// TIA Portal project "SortingStantion" (V16)
// Станция сортировки и отбраковки

(* hardware
DEVICE "S7-1200 station_1"  S7-1200 Station
   slot 0: "Rack_0"  S7-1200 Rack  Rack  V1.0
   slot 1: "6ES7 214-1AG40-0XB0"  CPU 1214C DC/DC/DC  6ES7 214-1AG40-0XB0  V4.4
*)

// ===== PLC "6ES7 214-1AG40-0XB0"  CPU 1214C DC/DC/DC =====

VAR_GLOBAL   // PLC tag table "Default tag table"
   "sensorFS1" AT %I200.0 : Bool;   // Фотодатчик 1
   "Tag_4" AT %IW0 : Word;
   "FS1" AT %I0.0 : Bool;   // Фотодатчик 1 (перед сканером)
   "GOOD_READ_SIGNAL" AT %I0.4 : Bool;   // Сигнал goodread
   "NO_READ_SIGNAL" AT %I0.3 : Bool;   // Сигнал NO_READ
   "FS2" AT %I0.1 : Bool;   // Фотодатчик перед отбраковщиком
   "FS3" AT %I0.2 : Bool;   // Фотодатчик на выходе отбраковщика
   "UPS_OK" AT %I0.5 : Bool;   // Статус ИБП - ОК
   "Conveyor_ON_impulse" AT %Q0.6 : Bool;
   "SCANER_PHASE_ON" AT %Q0.0 : Bool;   // Сингал для начала фазы сканирования
   "GreenLamp" AT %Q0.3 : Bool;
   "RedLamp" AT %Q0.4 : Bool;
   "PUSHER_OUT" AT %Q0.2 : Bool;
   "Buzzer" AT %Q0.5 : Bool;
   "Tag_6" AT %QW0 : Word;
   "SCANER_PHASE_OFF" AT %Q0.1 : Bool;   // Сигнал для окончания фазы сканирования
   "Conveyor_OFF_impulse" AT %Q0.7 : Bool;
   "Conveyor_ON_duplicate" AT %Q1.1 : Bool;
   "Tag_1" AT %M10.0 : Bool;
   "photoSensor0" AT %M0.0 : Bool;
   "sensorFS2" AT %M0.1 : Bool;
   "sensorFS3" AT %M0.2 : Bool;
   "System_Byte" AT %MB10 : Byte;
   "DiagStatusUpdate" AT %M10.1 : Bool;
   "AlwaysTRUE" AT %M10.2 : Bool;
   "AlwaysFALSE" AT %M10.3 : Bool;
   "Tag_2" AT %M2.0 : Bool;
   "Tag_3" AT %MD100 : DWord;
   "Tag_5" AT %MW0 : Word;
   "GoodRead" AT %M0.3 : Bool;
   "NoRead" AT %M0.4 : Bool;
   "Tag_7" AT %M1.3 : Bool;
   "Tag_8" AT %M1.4 : Bool;
   "FP_NEW_TASK" AT %M1.0 : Bool;
   "System" AT %M8.0 : Bool;
   "FN_MAIN_INTLK" AT %M8.1 : Bool;
   "FP_PHASE_ON" AT %M8.2 : Bool;
   "GoodReadTSignal" AT %M3.0 : Bool;
   "NoReadTSignal" AT %M3.1 : Bool;
   "wBuffer" AT %MW4 : Word;
   "HiChar" AT %MB4 : Byte;
   "loChar" AT %MB5 : Byte;
   "MEMMORYCELL_PRODUCT_DEFFECT_SETPOINT" AT %MD0 : DWord;
   "Tag_9" AT %M5.0 : Bool;
   "StrobeMerker" AT %M8.3 : Bool;
   "Control_begin" AT %M200.1 : Bool;   // Флаг запуска процесса контроля отбраковки
   "Tag_12" AT %M200.0 : Bool;
   "Tag_10" AT %MD170 : DInt;
   "TestMode" AT %M13.0 : Bool;
   "Clock_Byte" AT %MB65 : Byte;
   "Clock_10Hz" AT %M65.0 : Bool;
   "Clock_5Hz" AT %M65.1 : Bool;
   "Clock_2.5Hz" AT %M65.2 : Bool;
   "Clock_2Hz" AT %M65.3 : Bool;
   "Clock_1.25Hz" AT %M65.4 : Bool;
   "Clock_1Hz" AT %M65.5 : Bool;
   "Clock_0.625Hz" AT %M65.6 : Bool;
   "Clock_0.5Hz" AT %M65.7 : Bool;
   "Tag_14" AT %M13.1 : Bool;
   "Tag_15" AT %M13.2 : Bool;
   "Tag_16" AT %M13.3 : Bool;
   "Tag_17" AT %M13.4 : Bool;
   "Tag_19" AT %M64.0 : Bool;
   "Tag_20" AT %M13.5 : Bool;
   "Tag_21" AT %MB14 : Byte;
   "Tag_22" AT %MD14 : DWord;
   "Tag_23" AT %MD22 : DWord;
   "Tag_24" AT %M13.7 : Bool;
   "Tag_25" AT %MB11 : Byte;
   "Tag_26" AT %M13.6 : Bool;
   "Tag_27" AT %M198.6 : Bool;
   "Tag_11" AT %M8.4 : Bool;
   "FP_ERR_TRANSMITION" AT %M8.5 : Bool;
   "Tag_13" AT %M25.0 : Bool;
   "Tag_28" AT %M25.1 : Bool;
   "Флаг начала работы толкателя" AT %M25.2 : Bool;
   "Conveyor_ON" AT %Q1.0 : Bool;
END_VAR

TYPE "PRODUCT"
VERSION : 0.1
   STRUCT
      IS_ACTUAL : Bool := false;   // Флаг, указывающий на актуальность данных
      IS_GOOD : Bool;   // Флаг, указывающий то, что отбраковка не нужна
      ID : UDInt;   // Позиция в очереди
      BARCODE : String[100];   // Штрихкод из сканера в виде массива байт
      "TIME" : DTL;   // Метка времени
   END_STRUCT;
END_TYPE

DATA_BLOCK "GlobalData"   // DB1
{ S7_Optimized_Access := 'FALSE' }
VERSION : 0.1
   VAR
      INTERLOCK : Struct
         RESET_COUNTER_DISCONNECT : Bool;   // Команда для сброса счетчика, определяющего потерб связи с ПК
         MAIN_INTERLOCK : Bool;   // Главная деблокировка
         ACTIVE_ALARMS : Bool;   // Флаг, указывающий на наличае хотя бы одной ошибки
         DISCONNECT_COUNTER : UInt;   // Счетчик, по которому определяется потеря связи с ПК
         SPARE : Array[0..10] of Byte;
      END_STRUCT;
      AUX : Struct
         COUNTERS : Struct   // Счетчики заготовок
            QUANTITY_PRODUCTS : UDInt;   // Общее количество изделий, пройденых по конвейеру
            QUANTITY_BOXS : UDInt;   // Счетчик коробов
            QUANTITY_PRODUCTS_AUTO_REJECTED : UDInt;   // Количество изделий, отбракованых отбраковщиком автоматически
            QUANTITY_PRODUCTS_MANUAL_REJECTED : UDInt;   // Количество изделий, отбракованых вручную
            DEFECT_COUNTER : UDInt;   // Счетчик дефектного продукта
            REPEAT_COUNTER : UDInt;   // Счетчик повторов кодов
            SPARE : Array[0..22] of Word;
         END_STRUCT;
         BUZZER_ACTIVATE : Bool;   // Флаг активации звукового извещателя
         CONVEYOR_IS_STOPPED : Bool;   // Флаг, указывающий, что конвейер остановлен
         SPARE : Array[0..9] of Byte;
      END_STRUCT;
      FROM_HMI : Struct
         CTW : Struct   // Слово управления
            AUX_RUN_CMD : Bool;   // Команда для работы из PC
            RESET_ALARMS_CMD : Bool;   // Команда для сброса ошибок
            CLER_COLLECTION_CMD : Bool;   // Команда для очистки очереди изделий между отбраковщиком и сканером
            SIM_MODE_ACTIVE : Bool;   // Команда для активации режима симуляции
            CONVEYOR_FORCE_RUN : Bool;   // Команда для принудительного запуска конвейера
            HMI_IS_RUN : Bool;
            RUN_CMD_FROM_HMI : Bool;
            SPARE : Byte;
         END_STRUCT;
         SETTINGS : Struct   // Настройки панели
            IGNORE_REPEAT_PRODUCT_CODE_1 : Bool;   // Команда для игнорирования повтора кода продукта
            TIME_A : Time := T#5s;   // Задержка включения сканера, ms
            TIME_B : Time := T#5s;   // Длительность фазы чтения штрихкода, ms
            TIME_C : Time := T#5s;   // Время ожидания результа от сканера
            TIME_D : Time := T#4s;   // Длительность фазы чтения штрихкода, ms
            TIME_PUSHER_ACTIVE : Time := T#5s;   // Длительность импульса толкателя
            TIME_E : Time := T#5s;   // Время контроля отбраковки
            STOP_DELAY : Time := T#5s;   // Задержка остановки
            PRODUCT_DEFFECT_SETPOINT : UDInt := 5;   // Массовый брак (уставка)
            IGNORE_REPEAT_PRODUCT_CODE : Bool;   // Команда для игнорирования повтора кода продукта
            DEAD_TIME : Time := T#0ms;
            SPARE : Array[0..6] of Byte;
         END_STRUCT;
         CURRENT_TASK : Struct   // Текущее задание
            IN_WORK : Bool;   // Флаг, указывающий, что задание нахожится в работе
            ID : String[40];   // Уникальный идентификатор задания
            GTIN : String[40];   // Номер GTIN. (14 символов)
            PRODUCT_NAME : String[82];   // Наименование продукта
            LOT_NO : String[40];   // Номер производственной серии (до 20 символов)
            LINE_NUM : UInt := 0;   // Номер линии для, которой сформировано это задание.
            NUM_PACKS_IN_BOX : UDInt := 0;   // Кол-во продуктов в коробе.
            NUM_PACKS_IN_SERIES : UDInt := 0;   // Ожидаемое количество продуктов в серии (определяется по заданию на производство серии)
         END_STRUCT;
         SPARE : Array[0..6] of Byte;
      END_STRUCT;
      TO_HMI : Struct
         READ_PRODUCT_CMD : Bool;   // Команда для считывания данных продукта
      END_STRUCT;
      PRODUCT_IS_SCANING_AREA : "PRODUCT";   // Продукт в зоне сканирования
      PRODUCT_IS_PUSHER_AREA : "PRODUCT";   // Продукт в зоне отбраковки
      RESULT_STR : String;
      RCV_PRODUCT_ID : UDInt;   // ID продукта, полученного из L2 rкак подтверждение получения
   END_VAR
BEGIN
END_DATA_BLOCK

// folder: 10_ForTest

DATA_BLOCK "TestCodesGenerate_DB"   // DB25
{ S7_Optimized_Access := 'TRUE' }
VERSION : 0.1
// stored: InstanceOfName TestCodesGenerate
"TestCodesGenerate"
BEGIN
END_DATA_BLOCK

DATA_BLOCK "TestDB"   // DB26
{ S7_Optimized_Access := 'TRUE' }
VERSION : 0.1
   VAR
      Test_products : Array[0..1] of String[10];
      Test_disable_flag : Bool;
      Index_for_testproduct : UDInt;
      Actual_testproduct : String[50];
      counter_transfer_products : UDInt;
   END_VAR
BEGIN
   // Test_products[0] : Test_products
END_DATA_BLOCK

// folder: 2_КОНВЕЙЕР

DATA_BLOCK "CONVEYOR_DB"   // DB3
{ S7_Optimized_Access := 'TRUE' }
VERSION : 0.1
// stored: InstanceOfName CONVEYOR
"CONVEYOR"
BEGIN
END_DATA_BLOCK

// folder: 4_СКАНЕР MATRIX

DATA_BLOCK "SCANER_DB"   // DB2
{ S7_Optimized_Access := 'FALSE' }
VERSION : 0.1
// stored: InstanceOfName mSCANER
"mSCANER"
BEGIN
END_DATA_BLOCK

DATA_BLOCK "MODBUS_DATA"   // DB9
{ S7_Optimized_Access := 'FALSE' }
VERSION : 0.1
   VAR
      TCP_CONNECTION : TCON_IP_v4;
      MODBUS_DATA : Array[0..100] of Word;
      BYTES_ARRAY : Array[0..200] of Byte;
      Scaner_not_connected : Bool;
   END_VAR
BEGIN
   TCP_CONNECTION.ConnectionType := 11;
   TCP_CONNECTION.ID := 3;
   TCP_CONNECTION.InterfaceId := 64;
   TCP_CONNECTION.LocalPort := 502;
   TCP_CONNECTION.RemoteAddress.ADDR[1] := 0;
   TCP_CONNECTION.RemoteAddress.ADDR[2] := 0;
   TCP_CONNECTION.RemoteAddress.ADDR[3] := 0;
   TCP_CONNECTION.RemoteAddress.ADDR[4] := 0;
END_DATA_BLOCK

// folder: 5_ОТБРАКОВЩИК

DATA_BLOCK "PUSHER_CONTROL_DB"   // DB4
{ S7_Optimized_Access := 'TRUE' }
VERSION : 0.1
// stored: InstanceOfName PUSHER_CONTROL
"PUSHER_CONTROL"
BEGIN
END_DATA_BLOCK

DATA_BLOCK "PUSHER_DB_1"   // DB22
{ S7_Optimized_Access := 'TRUE' }
VERSION : 0.1
// stored: InstanceOfName PUSHER
"PUSHER"
BEGIN
END_DATA_BLOCK

// folder: 6_КОЛЛЕКЦИЯ ИЗДЕЛИЙ

DATA_BLOCK "ITEMS_COLLECTION"   // DB5
{ S7_Optimized_Access := 'FALSE' }
VERSION : 0.1
   VAR
      PRODUCTS_BEFOR_PUSHER : Struct
         LENGHT : UDInt;   // Количество изделий в коллекции
         INDEX : UDInt;   // Индекс для определения ID
         PRODUCTS : Array[0..20] of "PRODUCT";   // Коллекция невыпущенных продуктов
      END_STRUCT;
      PRODUCTS_IN_SEND_TO_PC : Struct
         LENGHT : UDInt;   // Количество изделий в коллекции
         INDEX : UDInt;   // Индекс для определения ID
         PRODUCTS : Array[0..3] of "PRODUCT";   // Коллекция продуктов в зоне отбраковщика
      END_STRUCT;
   END_VAR
BEGIN
END_DATA_BLOCK

// folder: 7_СООБЩЕНИЯ

DATA_BLOCK "ALARMS"   // DB6
{ S7_Optimized_Access := 'FALSE' }
VERSION : 0.1
   VAR
      WARNINGS : Struct
         WARNINGS_W0 : Word;   // Тэг для HMI
         WARNINGS_W1 : Word;   // Тэг для HMI
         WARNING_0_TASK_NOT_ACCEPTED : Bool;   // Сообщение - Задача не принята
         spare_1 : Bool;
         spare_2 : Bool;
         spare_3 : Bool;
         spare_4 : Bool;
         spare_5 : Bool;
         spare_6 : Bool;
         spare_7 : Bool;
         spare_8 : Bool;
         spare_9 : Bool;
         spare_10 : Bool;
         spare_11 : Bool;
         spare_12 : Bool;
         spare_13 : Bool;
         spare_14 : Bool;
         spare_15 : Bool;
         spare_16 : Bool;
         spare_17 : Bool;
         spare_18 : Bool;
         spare_19 : Bool;
         spare_20 : Bool;
         spare_21 : Bool;
         spare_22 : Bool;
         spare_23 : Bool;
         spare_24 : Bool;
         spare_25 : Bool;
         spare_26 : Bool;
         spare_27 : Bool;
         spare_28 : Bool;
         spare_29 : Bool;
         spare_30 : Bool;
         spare_31 : Bool;
      END_STRUCT;
      ALARMS : Struct
         ALARMS_W0 : Word;   // Тэг для HMI
         ALARMS_W1 : Word;   // Тэг для HMI
         ERROR_1_FS1_FAULT : Bool;   // Неисправность фотодатчика 1
         ERROR_2_FS2_FAULT : Bool;   // Неисправность фотодатчика 2
         ERROR_3_FS3_FAULT : Bool;   // Неисправность фотодатчика 3
         ERROR_4_REPEAT_PRODUCT_CODE : Bool;   // Повтор кода продукта
         ERROR_5_RECEIVING_CODE_WHEN_LINE_STOPS : Bool;   // Получение кода от сканера при остановке конвейера
         ERROR_6_ERROR_PUSHER : Bool;   // Ошибка отбраковщика (продукт не отбраковался)
         ERROR_7_OVER_DEFECT_COUNTER : Bool;   // Массовый брак
         ERROR_8_ERROR_TRANSMITIOM_BARCODE : Bool;   // Ошибка отбраковщика
         ERROR_9_ProductsAreTooCloseToEachOtherRangeScaner : Bool;   // Продукт слишком близко друг к другу
         ERROR_9_ProductsAreTooCloseToEachOtherRangePusher : Bool;
         ERROR_11_SPARE : Bool;
         ERROR_NO_TASK : Bool;   // Ошибка - нет принятой задачи
         ERROR_POWER_SYPLE : Bool;   // Ошибка питания (по сигналу от ИБП)
         ERROR_12_AutoScaner_NotConnected : Bool;
         spare_12 : Bool;
         spare_13 : Bool;
         spare_14 : Bool;
         spare_15 : Bool;
         spare_16 : Bool;
         spare_17 : Bool;
         spare_18 : Bool;
         spare_19 : Bool;
         spare_20 : Bool;
         spare_21 : Bool;
         spare_22 : Bool;
         spare_23 : Bool;
         spare_24 : Bool;
         spare_25 : Bool;
         spare_26 : Bool;
         spare_27 : Bool;
         spare_28 : Bool;
         spare_29 : Bool;
      END_STRUCT;
   END_VAR
BEGIN
END_DATA_BLOCK

// folder: 8_BUZZER

DATA_BLOCK "xBuzzer_DB"   // DB10
{ S7_Optimized_Access := 'TRUE' }
VERSION : 0.1
// stored: InstanceOfName xBuzzer
"xBuzzer"
BEGIN
END_DATA_BLOCK

// folder: 9_PINOUT

DATA_BLOCK "IO"   // DB15
{ S7_Optimized_Access := 'FALSE' }
VERSION : 0.1
   VAR
      INPUTS : Struct
         FS1 : Bool;
         FS2 : Bool;
         FS3 : Bool;
         GoodRead : Bool;
         NoRead : Bool;
         spare : Byte;
      END_STRUCT;
      OUTPUTS : Struct
         mScanerPhaseOn : Bool;
         mScanerPhaseOff : Bool;
         Pusher : Bool;
         GreenLamp : Bool;
         RedLamp : Bool;
         Buzzer : Bool;
         Conveyor : Bool;
         spare : Byte;
      END_STRUCT;
      SIMULATION : Struct
         FS1 : Bool;
         FS2 : Bool;
         FS3 : Bool;
         GoodRead : Bool;
         NoRead : Bool;
         spare : Byte;
      END_STRUCT;
   END_VAR
BEGIN
END_DATA_BLOCK

// folder: System blocks/Program resources

DATA_BLOCK "SDTIMER_ALARM_FS1"   // DB7
{ S7_Optimized_Access := 'TRUE' }
AUTHOR : Simatic
FAMILY : IEC
NAME : IEC_TMR
VERSION : 1.0
// stored: InstanceOfName IEC_TIMER
"IEC_TIMER"
BEGIN
END_DATA_BLOCK

DATA_BLOCK "SDTIMER_ALARM_FS2"   // DB11
{ S7_Optimized_Access := 'TRUE' }
AUTHOR : Simatic
FAMILY : IEC
NAME : IEC_TMR
VERSION : 1.0
// stored: InstanceOfName IEC_TIMER
"IEC_TIMER"
BEGIN
END_DATA_BLOCK

DATA_BLOCK "SDTIMER_ALARM_FS3"   // DB12
{ S7_Optimized_Access := 'TRUE' }
AUTHOR : Simatic
FAMILY : IEC
NAME : IEC_TMR
VERSION : 1.0
// stored: InstanceOfName IEC_TIMER
"IEC_TIMER"
BEGIN
END_DATA_BLOCK

DATA_BLOCK "IEC_Timer_0_DGR"   // DB13
{ S7_Optimized_Access := 'TRUE' }
AUTHOR : Simatic
FAMILY : IEC
NAME : IEC_TMR
VERSION : 1.0
// stored: InstanceOfName IEC_TIMER
"IEC_TIMER"
BEGIN
END_DATA_BLOCK

DATA_BLOCK "IEC_Timer_0_NR"   // DB14
{ S7_Optimized_Access := 'TRUE' }
AUTHOR : Simatic
FAMILY : IEC
NAME : IEC_TMR
VERSION : 1.0
// stored: InstanceOfName IEC_TIMER
"IEC_TIMER"
BEGIN
END_DATA_BLOCK

DATA_BLOCK "IEC_TIM_FS3"   // DB16
{ S7_Optimized_Access := 'TRUE' }
AUTHOR : Simatic
FAMILY : IEC
NAME : IEC_TMR
VERSION : 1.0
// stored: InstanceOfName IEC_TIMER
"IEC_TIMER"
BEGIN
END_DATA_BLOCK

DATA_BLOCK "#IEC_TIM_FS1"   // DB17
{ S7_Optimized_Access := 'TRUE' }
AUTHOR : Simatic
FAMILY : IEC
NAME : IEC_TMR
VERSION : 1.0
// stored: InstanceOfName IEC_TIMER
"IEC_TIMER"
BEGIN
END_DATA_BLOCK

DATA_BLOCK "#IEC_TIM_FS2"   // DB18
{ S7_Optimized_Access := 'TRUE' }
AUTHOR : Simatic
FAMILY : IEC
NAME : IEC_TMR
VERSION : 1.0
// stored: InstanceOfName IEC_TIMER
"IEC_TIMER"
BEGIN
END_DATA_BLOCK

DATA_BLOCK "IEC_TIM_PHASEOFF"   // DB19
{ S7_Optimized_Access := 'TRUE' }
AUTHOR : Simatic
FAMILY : IEC
NAME : IEC_TMR
VERSION : 1.0
// stored: InstanceOfName IEC_TIMER
"IEC_TIMER"
BEGIN
END_DATA_BLOCK

DATA_BLOCK "IEC_Timer_0_DB_1"   // DB20
{ S7_Optimized_Access := 'TRUE' }
AUTHOR : Simatic
FAMILY : IEC
NAME : IEC_TMR
VERSION : 1.0
// stored: InstanceOfName IEC_TIMER
"IEC_TIMER"
BEGIN
END_DATA_BLOCK

DATA_BLOCK "SD_TIMER"   // DB21
{ S7_Optimized_Access := 'TRUE' }
AUTHOR : Simatic
FAMILY : IEC
NAME : IEC_TMR
VERSION : 1.0
// stored: InstanceOfName IEC_TIMER
"IEC_TIMER"
BEGIN
END_DATA_BLOCK

DATA_BLOCK "IEC_Timer_0_DB"   // DB23
{ S7_Optimized_Access := 'TRUE' }
AUTHOR : Simatic
FAMILY : IEC
NAME : IEC_TMR
VERSION : 1.0
// stored: InstanceOfName IEC_TIMER
"IEC_TIMER"
BEGIN
END_DATA_BLOCK

DATA_BLOCK "IEC_Timer_0_DB_2"   // DB24
{ S7_Optimized_Access := 'TRUE' }
AUTHOR : Simatic
FAMILY : IEC
NAME : IEC_TMR
VERSION : 1.0
// stored: InstanceOfName IEC_TIMER
"IEC_TIMER"
BEGIN
END_DATA_BLOCK

DATA_BLOCK "ADDR_SEND_UDP"   // DB29
{ S7_Optimized_Access := 'TRUE' }
   VAR
      ConnectionData : TCON_IP_v4;
      ADDR_Send : TADDR_Param;
   END_VAR
BEGIN
   ConnectionData.ID := 1;
   ConnectionData.ConnectionType := 19;
   ConnectionData.InterfaceId := 64;
   ConnectionData.LocalPort := 2000;
   ConnectionData.RemotePort := 0;
   ConnectionData.ActiveEstablished := false;
   ADDR_Send.REM_PORT_NR := 2000;
   ADDR_Send.REM_IP_ADDR[1] := 192;
   ADDR_Send.REM_IP_ADDR[2] := 168;
   ADDR_Send.REM_IP_ADDR[3] := 3;
   ADDR_Send.REM_IP_ADDR[4] := 97;
END_DATA_BLOCK

DATA_BLOCK "_6ES7 214-1AG40-0XB0_Receive_DB"   // DB30
{ S7_Optimized_Access := 'TRUE' }
   VAR
      ConnectionData : TCON_IP_v4;
      ADDR_Send : TADDR_Param;
   END_VAR
BEGIN
   ConnectionData.ID := 4;
   ConnectionData.ConnectionType := 19;
   ConnectionData.InterfaceId := 64;
   ConnectionData.LocalPort := 2002;
   ConnectionData.RemotePort := 0;
   ConnectionData.ActiveEstablished := false;
   ADDR_Send.REM_PORT_NR := 0;
END_DATA_BLOCK

DATA_BLOCK "ADDR_RCV_UDP"   // DB31
{ S7_Optimized_Access := 'TRUE' }
   VAR
      ConnectionData : TCON_IP_v4;
      ADDR_Send : TADDR_Param;
   END_VAR
BEGIN
   ConnectionData.ID := 2;
   ConnectionData.ConnectionType := 19;
   ConnectionData.InterfaceId := 64;
   ConnectionData.LocalPort := 2001;
   ConnectionData.RemotePort := 0;
   ConnectionData.ActiveEstablished := false;
   ADDR_Send.REM_PORT_NR := 0;
   ADDR_Send.REM_IP_ADDR[1] := 0;
   ADDR_Send.REM_IP_ADDR[2] := 0;
   ADDR_Send.REM_IP_ADDR[3] := 0;
   ADDR_Send.REM_IP_ADDR[4] := 0;
END_DATA_BLOCK

DATA_BLOCK "IEC_Timer_0_DB_3"   // DB32
{ S7_Optimized_Access := 'TRUE' }
AUTHOR : Simatic
FAMILY : IEC
NAME : IEC_TMR
VERSION : 1.0
// stored: InstanceOfName IEC_TIMER
"IEC_TIMER"
BEGIN
END_DATA_BLOCK

// folder: (top level)

ORGANIZATION_BLOCK "Main"   // OB1, LAD, ProgramCycle
TITLE = "Main Program Sweep (Cycle)"
{ S7_Optimized_Access := 'TRUE' }
VERSION : 0.1
   VAR_INPUT
      Initial_Call : Bool;   // Initial call of this OB
      Remanence : Bool;   // =True, if remanent data are available
   END_VAR
   VAR_TEMP
      LineIsRunNormalMode : Bool;   // Флаг, указывающий, что линия запущена в нормальном режиме
      LineRunEnable : Bool;   // Флаг, разрешающий работу линии
      ScanerStage : Word;
      PusherControlStage : Word;
      PusherStage : Word;
   END_VAR
BEGIN

REGION Network 1: Главная деблокировка
   // Проверка разрешения для работы установки
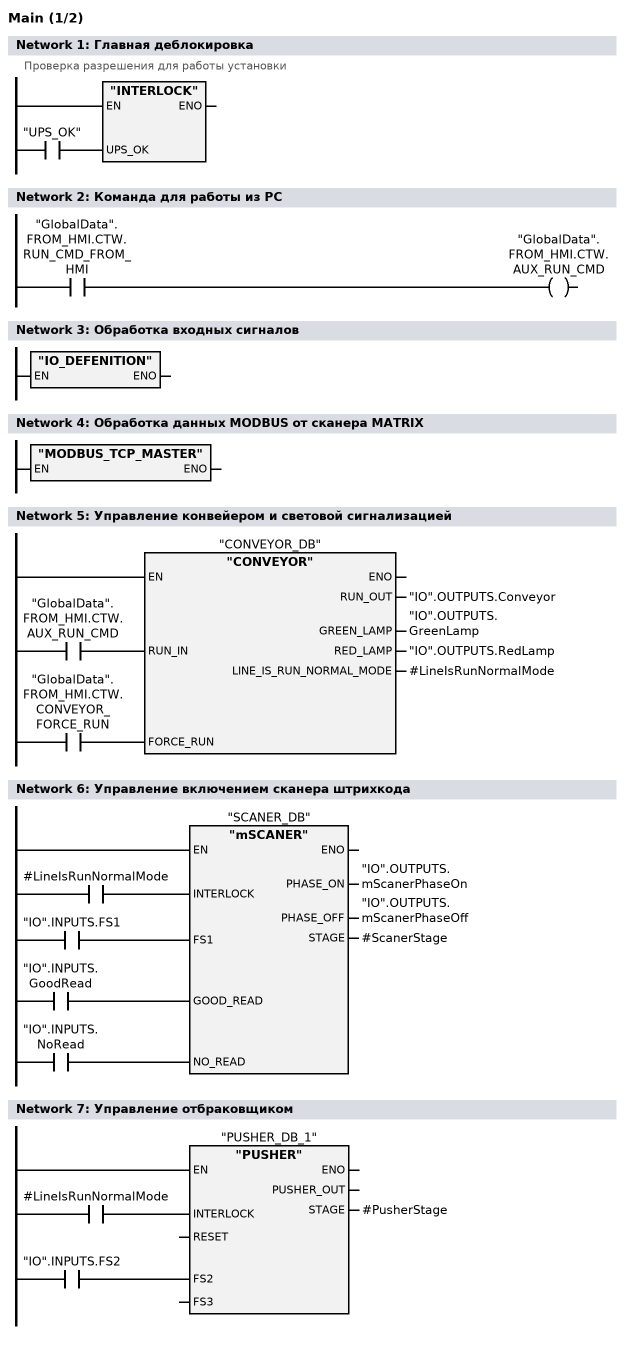
   RUNG wire#powerrail
      "INTERLOCK"(UPS_OK := wire#w1)
   END_RUNG
   RUNG wire#powerrail
      Contact( "UPS_OK" )
   END_RUNG wire#w1
   // the same network as SCL:
   "INTERLOCK"(UPS_OK := "UPS_OK");
END_REGION

REGION Network 2: Команда для работы из PC
   RUNG wire#powerrail
      Contact( "GlobalData".FROM_HMI.CTW.RUN_CMD_FROM_HMI )
      Coil( "GlobalData".FROM_HMI.CTW.AUX_RUN_CMD )
   END_RUNG
   // the same network as SCL:
   "GlobalData".FROM_HMI.CTW.AUX_RUN_CMD := "GlobalData".FROM_HMI.CTW.RUN_CMD_FROM_HMI;
END_REGION

REGION Network 3: Обработка входных сигналов
   RUNG wire#powerrail
      "IO_DEFENITION"()
   END_RUNG
   // the same network as SCL:
   "IO_DEFENITION"();
END_REGION

REGION Network 4: Обработка данных MODBUS от сканера MATRIX
   RUNG wire#powerrail
      "MODBUS_TCP_MASTER"()
   END_RUNG
   // the same network as SCL:
   "MODBUS_TCP_MASTER"();
END_REGION

REGION Network 5: Управление конвейером и световой сигнализацией
   RUNG wire#powerrail
      "CONVEYOR_DB"(RUN_IN := wire#w1, FORCE_RUN := wire#w2, RUN_OUT => "IO".OUTPUTS.Conveyor, GREEN_LAMP => "IO".OUTPUTS.GreenLamp, RED_LAMP => "IO".OUTPUTS.RedLamp, LINE_IS_RUN_NORMAL_MODE => #LineIsRunNormalMode)
   END_RUNG
   RUNG wire#powerrail
      Contact( "GlobalData".FROM_HMI.CTW.AUX_RUN_CMD )
   END_RUNG wire#w1
   RUNG wire#powerrail
      Contact( "GlobalData".FROM_HMI.CTW.CONVEYOR_FORCE_RUN )
   END_RUNG wire#w2
   // the same network as SCL:
   "CONVEYOR_DB"(RUN_IN := "GlobalData".FROM_HMI.CTW.AUX_RUN_CMD,   // "CONVEYOR"
                 FORCE_RUN := "GlobalData".FROM_HMI.CTW.CONVEYOR_FORCE_RUN,
                 RUN_OUT => "IO".OUTPUTS.Conveyor,
                 GREEN_LAMP => "IO".OUTPUTS.GreenLamp,
                 RED_LAMP => "IO".OUTPUTS.RedLamp,
                 LINE_IS_RUN_NORMAL_MODE => #LineIsRunNormalMode);
END_REGION

REGION Network 6: Управление включением сканера штрихкода
   RUNG wire#powerrail
      "SCANER_DB"(INTERLOCK := wire#w1, FS1 := wire#w2, GOOD_READ := wire#w3, NO_READ := wire#w4, PHASE_ON => "IO".OUTPUTS.mScanerPhaseOn, PHASE_OFF => "IO".OUTPUTS.mScanerPhaseOff, STAGE => #ScanerStage)
   END_RUNG
   RUNG wire#powerrail
      Contact( #LineIsRunNormalMode )
   END_RUNG wire#w1
   RUNG wire#powerrail
      Contact( "IO".INPUTS.FS1 )
   END_RUNG wire#w2
   RUNG wire#powerrail
      Contact( "IO".INPUTS.GoodRead )
   END_RUNG wire#w3
   RUNG wire#powerrail
      Contact( "IO".INPUTS.NoRead )
   END_RUNG wire#w4
   // the same network as SCL:
   "SCANER_DB"(INTERLOCK := #LineIsRunNormalMode,   // "mSCANER"
               FS1 := "IO".INPUTS.FS1,
               GOOD_READ := "IO".INPUTS.GoodRead,
               NO_READ := "IO".INPUTS.NoRead,
               PHASE_ON => "IO".OUTPUTS.mScanerPhaseOn,
               PHASE_OFF => "IO".OUTPUTS.mScanerPhaseOff,
               STAGE => #ScanerStage);
END_REGION

REGION Network 7: Управление отбраковщиком
   RUNG wire#powerrail
      "PUSHER_DB_1"(INTERLOCK := wire#w1, FS2 := wire#w2, RESET :=, FS3 :=, PUSHER_OUT =>, STAGE => #PusherStage)
   END_RUNG
   RUNG wire#powerrail
      Contact( #LineIsRunNormalMode )
   END_RUNG wire#w1
   RUNG wire#powerrail
      Contact( "IO".INPUTS.FS2 )
   END_RUNG wire#w2
   // the same network as SCL:
   "PUSHER_DB_1"(INTERLOCK := #LineIsRunNormalMode, FS2 := "IO".INPUTS.FS2, STAGE => #PusherStage);   // "PUSHER"
END_REGION

REGION Network 8: Задвигание толкателя
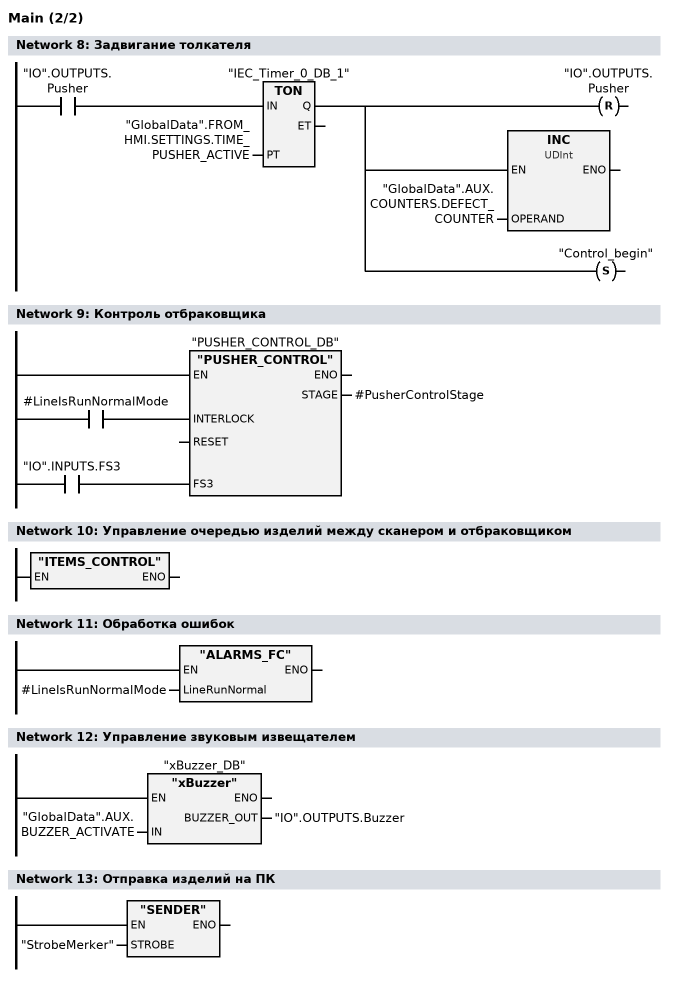
   "IEC_Timer_0_DB_1".TON(IN := "IO".OUTPUTS.Pusher, PT := "GlobalData".FROM_HMI.SETTINGS.TIME_PUSHER_ACTIVE);
   IF "IEC_Timer_0_DB_1".Q THEN
       "IO".OUTPUTS.Pusher := FALSE;
       "GlobalData".AUX.COUNTERS.DEFECT_COUNTER := "GlobalData".AUX.COUNTERS.DEFECT_COUNTER + 1;
       "Control_begin" := TRUE;
   END_IF;
END_REGION

REGION Network 9: Контроль отбраковщика
   RUNG wire#powerrail
      "PUSHER_CONTROL_DB"(INTERLOCK := wire#w1, FS3 := wire#w2, RESET :=, STAGE => #PusherControlStage)
   END_RUNG
   RUNG wire#powerrail
      Contact( #LineIsRunNormalMode )
   END_RUNG wire#w1
   RUNG wire#powerrail
      Contact( "IO".INPUTS.FS3 )
   END_RUNG wire#w2
   // the same network as SCL:
   "PUSHER_CONTROL_DB"(INTERLOCK := #LineIsRunNormalMode, FS3 := "IO".INPUTS.FS3, STAGE => #PusherControlStage);   // "PUSHER_CONTROL"
END_REGION

REGION Network 10: Управление очередью изделий между сканером и отбраковщиком
   RUNG wire#powerrail
      "ITEMS_CONTROL"()
   END_RUNG
   // the same network as SCL:
   "ITEMS_CONTROL"();
END_REGION

REGION Network 11: Обработка ошибок
   RUNG wire#powerrail
      "ALARMS_FC"(LineRunNormal := #LineIsRunNormalMode)
   END_RUNG
   // the same network as SCL:
   "ALARMS_FC"(LineRunNormal := #LineIsRunNormalMode);
END_REGION

REGION Network 12: Управление звуковым извещателем
   RUNG wire#powerrail
      "xBuzzer_DB"(IN := "GlobalData".AUX.BUZZER_ACTIVATE, BUZZER_OUT => "IO".OUTPUTS.Buzzer)
   END_RUNG
   // the same network as SCL:
   "xBuzzer_DB"(IN := "GlobalData".AUX.BUZZER_ACTIVATE, BUZZER_OUT => "IO".OUTPUTS.Buzzer);   // "xBuzzer"
END_REGION

REGION Network 13: Отправка изделий на ПК
   RUNG wire#powerrail
      "SENDER"(STROBE := "StrobeMerker")
   END_RUNG
   // the same network as SCL:
   "SENDER"(STROBE := "StrobeMerker");
END_REGION
END_ORGANIZATION_BLOCK

ORGANIZATION_BLOCK "Cyclic interrupt"   // OB30, SCL, CyclicInterrupt
{ S7_Optimized_Access := 'TRUE' }
VERSION : 0.1
   VAR_INPUT
      Initial_Call : Bool;   // Initial call of this OB
      Event_Count : Int;   // Events discarded
   END_VAR
BEGIN
   //Если отсутсвует деблокировка, то смысла инкриментировать счетчик
   //по которому определяется разрыв связи с ПК нет
   IF "GlobalData".INTERLOCK.MAIN_INTERLOCK = FALSE THEN
       RETURN;
   END_IF;

   //Инкрементация счетчика, по которому определяется разрыв 
   //соединения с ПК
   "GlobalData".INTERLOCK.DISCONNECT_COUNTER := "GlobalData".INTERLOCK.DISCONNECT_COUNTER + 1;
END_ORGANIZATION_BLOCK

ORGANIZATION_BLOCK "Cyclic interrupt_5MS"   // OB31, LAD, CyclicInterrupt
{ S7_Optimized_Access := 'TRUE' }
VERSION : 0.1
   VAR_INPUT
      Initial_Call : Bool;   // Initial call of this OB
      Event_Count : Int;   // Events discarded
   END_VAR
BEGIN

REGION Network 1
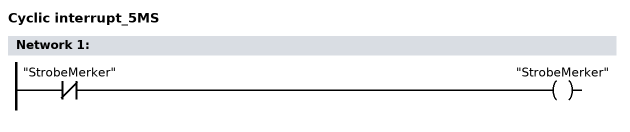
   RUNG wire#powerrail
      I_Contact( "StrobeMerker" )
      Coil( "StrobeMerker" )
   END_RUNG
   // the same network as SCL:
   "StrobeMerker" := NOT "StrobeMerker";
END_REGION
END_ORGANIZATION_BLOCK

ORGANIZATION_BLOCK "Startup"   // OB100, LAD, Startup
TITLE = "Complete Restart"
{ S7_Optimized_Access := 'TRUE' }
VERSION : 0.1
   VAR_INPUT
      LostRetentive : Bool;   // True if retentive data are lost
      LostRTC : Bool;   // True if date and time are lost
   END_VAR
BEGIN

REGION Network 1 (SCL): Запись значения из настройки МАССОВЫЙ БРАК в переменную
   "MEMMORYCELL_PRODUCT_DEFFECT_SETPOINT" := "GlobalData".FROM_HMI.SETTINGS.PRODUCT_DEFFECT_SETPOINT;
END_REGION
END_ORGANIZATION_BLOCK

// folder: 10_ForTest

FUNCTION_BLOCK "TestCodesGenerate"   // FB8, LAD
{ S7_Optimized_Access := 'TRUE' }
VERSION : 0.1
   VAR_INPUT
      index_for_testproduct : UDInt;
   END_VAR
   VAR
      CountChars : UInt;
      Array_of_chars : Array[0..33] of Byte;
   END_VAR
   // Array_of_chars[0] := 16#02;
   // Array_of_chars[1] := 16#30;
   // Array_of_chars[2] := 16#31;
   // Array_of_chars[3] := 16#30;
   // Array_of_chars[4] := 16#34;
   // Array_of_chars[5] := 16#36;
   // Array_of_chars[6] := 16#30;
   // Array_of_chars[7] := 16#34;
   // Array_of_chars[8] := 16#35;
   // Array_of_chars[9] := 16#36;
   // Array_of_chars[10] := 16#37;
   // Array_of_chars[11] := 16#38;
   // Array_of_chars[12] := 16#39;
   // Array_of_chars[13] := 16#30;
   // Array_of_chars[14] := 16#31;
   // Array_of_chars[15] := 16#32;
   // Array_of_chars[16] := 16#36;
   // Array_of_chars[17] := 16#32;
   // Array_of_chars[18] := 16#31;
   // Array_of_chars[19] := 16#24;
   // Array_of_chars[25] := 16#1D;
   // Array_of_chars[26] := 16#39;
   // Array_of_chars[27] := 16#33;
   // Array_of_chars[32] := 16#0D;
   // Array_of_chars[33] := 16#0A;
   // Array_of_chars[20] := 16#24;
   // Array_of_chars[21] := 16#24;
   // Array_of_chars[22] := 16#24;
   // Array_of_chars[23] := 16#24;
   // Array_of_chars[24] := 16#24;
   // Array_of_chars[28] := 16#24;
   // Array_of_chars[29] := 16#24;
   // Array_of_chars[30] := 16#24;
   // Array_of_chars[31] := 16#24;
BEGIN

REGION Network 1: Разбиваем строку с серийным кодом на символы utf-8 в формате байт и кладем их в заготовленный массив с неизменными символами кода (GTIN, криптохвост, идентификаторы полей и стандартные префиксы)
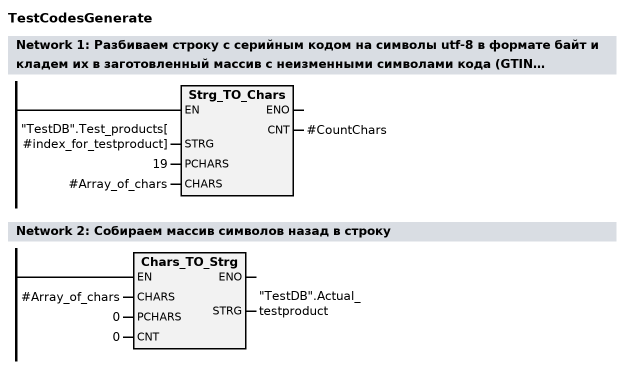
   // no SCL statement known for Strg_TO_Chars: written as a call
   Strg_TO_Chars(Strg := "TestDB".Test_products[#index_for_testproduct],
                 pChars := 19,
                 Chars := #Array_of_chars,
                 Cnt => #CountChars);
END_REGION

REGION Network 2: Собираем массив символов назад в строку
   // no SCL statement known for Chars_TO_Strg: written as a call
   Chars_TO_Strg(Chars := #Array_of_chars, pChars := 0, Cnt := 0, Strg => "TestDB".Actual_testproduct);
END_REGION

REGION Network 3 (SCL)
   // Увеличиваем счетчик тестовых продуктов и если перебор, то устанавливаем флаг запрета тестирования
   "TestDB".Index_for_testproduct := "TestDB".Index_for_testproduct + 1;
   IF "TestDB".Index_for_testproduct > 4999 THEN
       //"TestDB".Test_disable_flag := 1;
       "TestDB".Index_for_testproduct := 0;
   END_IF;
END_REGION
END_FUNCTION_BLOCK

// folder: 11_ОТПРАВКА В ПК

FUNCTION "SENDER" : Void   // FC1, LAD
{ S7_Optimized_Access := 'TRUE' }
VERSION : 0.1
   VAR_INPUT
      STROBE : Bool;   // Стробирующий сигнал
   END_VAR
   VAR_TEMP
      Index : UDInt;
      "Counter" : UDInt;
      Lenght : UDInt;
      send_cmd : Bool;
      doneSend : Bool;
      bysySend : Bool;
      errorSend : Bool;
      statusSend : Word;
      doneRecv : Bool;
      bysyRecv : Bool;
      errorRecv : Bool;
      statusRecv : Word;
      number_of_fail_of_done : Word;
      Header : String;
      ResultStr : String;
      ASK : Bool;
      ASK_BYTE : Byte;
      INDEX_STR : String;
      TimeOut : Bool;
   END_VAR
BEGIN

REGION Network 1: Получение ответа от L2 об успешно полученном штрихкоде
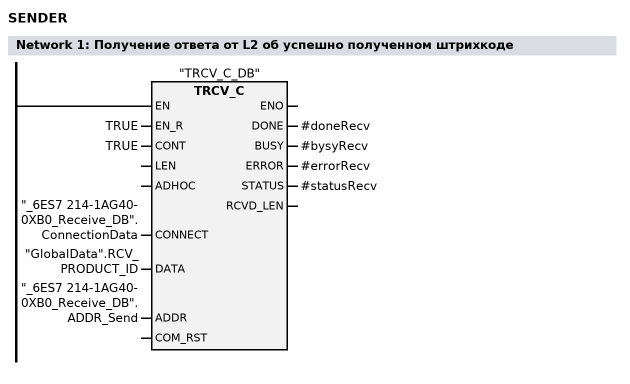
   "TRCV_C_DB"(EN_R := TRUE,   // TRCV_C
               CONT := TRUE,
               CONNECT := "_6ES7 214-1AG40-0XB0_Receive_DB".ConnectionData,
               DATA := "GlobalData".RCV_PRODUCT_ID,
               ADDR := "_6ES7 214-1AG40-0XB0_Receive_DB".ADDR_Send,
               DONE => #doneRecv,
               BUSY => #bysyRecv,
               ERROR => #errorRecv,
               STATUS => #statusRecv);
END_REGION

REGION Network 2 (SCL): В случае отсутсвия продуктов в коллнеции на передачу - выход
   IF "ITEMS_COLLECTION".PRODUCTS_IN_SEND_TO_PC.LENGHT = 0 THEN
       RETURN;
   END_IF;
END_REGION

REGION Network 3 (SCL): Форматирование строки
   //Добавление к строке ключа ID
   "GlobalData".RESULT_STR := 'ID=';

   //Поличение значения ID в текстовом виде
   "UDINT_TO_STR"(IN := "ITEMS_COLLECTION".PRODUCTS_IN_SEND_TO_PC.PRODUCTS[0].ID,
                  OUT => #INDEX_STR);

   //Добавление к строке значения ID
   "GlobalData".RESULT_STR := CONCAT(IN1 := "GlobalData".RESULT_STR,
                                     IN2 := #INDEX_STR);

   //Добавление к строке ключа BARCODE
   "GlobalData".RESULT_STR := CONCAT(IN1 := "GlobalData".RESULT_STR,
                                     IN2 := '   BARCODE=');

   //Добавление к строке значения BARCODE
   "GlobalData".RESULT_STR := CONCAT(IN1 := "GlobalData".RESULT_STR,
                                     IN2 := "ITEMS_COLLECTION".PRODUCTS_IN_SEND_TO_PC.PRODUCTS[0].BARCODE);
END_REGION

REGION Network 4 (SCL): Отправка штрихкода на L2 по UDP каналу
   // Отправка выполняется по стобирующему сигналу STROBE
   "TSEND_C_UDP"(REQ:=#STROBE,
                 CONT:=TRUE,
                 DONE=>#doneSend,
                 BUSY=>#bysySend,
                 ERROR=>#errorSend,
                 STATUS=>#statusSend,
                 CONNECT:="ADDR_SEND_UDP".ConnectionData,
                 DATA:="GlobalData".RESULT_STR,
                 ADDR:="ADDR_SEND_UDP".ADDR_Send);
END_REGION

REGION Network 5 (SCL): Формирование бита подтверждения
   // Если от L2 получен ответ 255, тогда ASK=TRUE
   #ASK := "GlobalData".RCV_PRODUCT_ID = "ITEMS_COLLECTION".PRODUCTS_IN_SEND_TO_PC.PRODUCTS[0].ID;
END_REGION

REGION Network 6 (SCL): При получении бита подтверждениясмещаем коллекцию вверх
   IF #ASK = TRUE THEN

       #Counter := 0;
       #Lenght := "ITEMS_COLLECTION".PRODUCTS_IN_SEND_TO_PC.#LENGHT;

       //Стираем данные из самой верхней
       //ячейки
       "ITEMS_COLLECTION".PRODUCTS_IN_SEND_TO_PC.PRODUCTS[0].IS_ACTUAL := FALSE;
       "ITEMS_COLLECTION".PRODUCTS_IN_SEND_TO_PC.PRODUCTS[0].BARCODE := '';
       "ITEMS_COLLECTION".PRODUCTS_IN_SEND_TO_PC.PRODUCTS[0].IS_GOOD := FALSE;


       //Цикл, в котором переносятся активные 
       //данные
       FOR #Index := 1 TO #Lenght DO

           IF "ITEMS_COLLECTION".PRODUCTS_IN_SEND_TO_PC.PRODUCTS[#Index].IS_ACTUAL = TRUE THEN

               //Перемещение данных из временной коллекции в постояную
               "ITEMS_COLLECTION".PRODUCTS_IN_SEND_TO_PC.PRODUCTS[#Counter] := "ITEMS_COLLECTION".PRODUCTS_IN_SEND_TO_PC.PRODUCTS[#Index];

               //Инкрементация счетчика
               #Counter := #Counter + 1;

               CONTINUE;

           END_IF;

       END_FOR;

       //Цикл в котором все оставшиеся данные затираются
       FOR #Index := #Counter TO 3 DO

           "ITEMS_COLLECTION".PRODUCTS_IN_SEND_TO_PC.PRODUCTS[#Index].IS_ACTUAL := FALSE;
           "ITEMS_COLLECTION".PRODUCTS_IN_SEND_TO_PC.PRODUCTS[#Index].BARCODE := '';
           "ITEMS_COLLECTION".PRODUCTS_IN_SEND_TO_PC.PRODUCTS[#Index].ID := 0;
           "ITEMS_COLLECTION".PRODUCTS_IN_SEND_TO_PC.PRODUCTS[#Index].IS_GOOD := FALSE;

       END_FOR;

       //Передача количества изделий
       "ITEMS_COLLECTION".PRODUCTS_IN_SEND_TO_PC.LENGHT := #Counter;


   END_IF;
END_REGION

REGION Network 7 (SCL): Формирования ошибки ожидания результата подтверждения от L2
   IF "ITEMS_COLLECTION".PRODUCTS_IN_SEND_TO_PC.LENGHT > 2 THEN
       "ALARMS".ALARMS.ERROR_8_ERROR_TRANSMITIOM_BARCODE := TRUE;
   END_IF;
END_REGION
END_FUNCTION

// folder: 12_Unknown

FUNCTION_BLOCK "frontPositive"   // FB3, SCL
{ S7_Optimized_Access := 'TRUE' }
VERSION : 0.1
   VAR_INPUT
      INPUT : Bool;
   END_VAR
   VAR_OUTPUT
      RESULT : Bool;   // Результат выполнения блока
   END_VAR
   VAR
      OLD_STATE : Bool;   // Старое значение
   END_VAR
BEGIN
   (*
       ФУНКЦИОНАЛЬНЫЙ БЛОК, ПРЕДНАЗНАЧЕНЫЙ ДЛЯ ВЫДЕЛЕНИЯ
       ПОЛОЖИТЕЛЬНОГО ФРОНТА СИГНАЛА
   *)

   //Проверка на определение положительного
   //фронта сигнала
   #RESULT := (#INPUT = true AND #OLD_STATE = FALSE);

   //Запоминаем состояние сигнала
   #OLD_STATE := #INPUT;
END_FUNCTION_BLOCK

FUNCTION_BLOCK "Timer"   // FB4, SCL
{ S7_Optimized_Access := 'TRUE' }
VERSION : 0.1
   VAR_INPUT
      Enable : Bool;
      "Time" : UInt;
   END_VAR
   VAR_OUTPUT
      Result : Bool;
   END_VAR
   VAR_IN_OUT
      t0 : TON_TIME;
   END_VAR
BEGIN
END_FUNCTION_BLOCK

FUNCTION "COMPARE_GTIN" : Bool   // FC4, LAD
TITLE = Сравнение GTIN
{ S7_Optimized_Access := 'TRUE' }
VERSION : 0.1
   VAR_INPUT
      GTIN_FROM_TASK : String;
      GTIN_FROM_SCAN_RESULT_1 : String;
   END_VAR
   VAR_TEMP
      CHARS_FROM_TASK : Array[0..40] of Char;
      CHARS_FROM_TASK_LENGHT : Int;
      CHARS_FROM_SCAN_RESULT : Array[0..40] of Char;
      CHARS_FROM_SCAN_RESULT_LENGHT : Int;
      CONTER : Int;
   END_VAR
BEGIN

REGION Network 1 (SCL): Получение символов из GTIN задания
   Strg_TO_Chars(Strg:=#GTIN_FROM_TASK,
                 pChars:=0,
                 Cnt=>#CHARS_FROM_TASK_LENGHT,
                 Chars:=#CHARS_FROM_TASK);
END_REGION

REGION Network 2 (SCL): Получение символов из GTIN результата сканирования
   Strg_TO_Chars(Strg := #GTIN_FROM_SCAN_RESULT_1,
                 pChars := 0,
                 Cnt => #CHARS_FROM_SCAN_RESULT_LENGHT,
                 Chars := #CHARS_FROM_SCAN_RESULT);
END_REGION

REGION Network 3 (SCL): Сравнение длины строк
   // Если длина обеих строк не равна, возвращаем FALSE
   IF #CHARS_FROM_TASK_LENGHT <> #CHARS_FROM_SCAN_RESULT_LENGHT THEN

       //Устанавливаем результат выполнения функции
       #COMPARE_GTIN := FALSE;

       //Устанавливаем ошибке
       "ALARMS".ALARMS.ERROR_1_FS1_FAULT := TRUE;

       //Выход из функции
       RETURN;
   END_IF;
END_REGION

REGION Network 4 (SCL): Посимвольное сравнение строк
   FOR #CONTER := 0 TO #CHARS_FROM_TASK_LENGHT DO

       IF #CHARS_FROM_TASK[#CONTER] <> #CHARS_FROM_SCAN_RESULT[#CONTER] THEN

           //Устанавливаем результат выполнения функции
           #COMPARE_GTIN := FALSE;

           //Устанавливаем ошибке
           "ALARMS".ALARMS.ERROR_1_FS1_FAULT := TRUE;

           //Выход из функции
           RETURN;

       END_IF;

   END_FOR;
END_REGION

REGION Network 5 (SCL): Возврат результата сравнения TRUE
   // Если ранее из функции не вышли, значит строки одинаковые.
   //Устанавливаем результат выполнения функции
   #COMPARE_GTIN := TRUE;

   //Выход из функции
   RETURN;
END_REGION
END_FUNCTION

FUNCTION "RESERVATOIN" : Void   // FC5, SCL
{ S7_Optimized_Access := 'TRUE' }
VERSION : 0.1
BEGIN
   (*
       ЛОКАЛЬНЫЙ МЕТОД
       РЕЗЕРВИРОВАНИЕ МЕСТА ПОД НОВОЕ ИЗДЕЛИЕ  

       резервируем место в конце коллекции,
       для того, чтоб записать туда данные, полученые от сканера
   *)

   "ITEMS_COLLECTION".PRODUCTS_BEFOR_PUSHER.PRODUCTS ["ITEMS_COLLECTION".PRODUCTS_BEFOR_PUSHER.LENGHT].IS_GOOD := FALSE;
   "ITEMS_COLLECTION".PRODUCTS_BEFOR_PUSHER.PRODUCTS["ITEMS_COLLECTION".PRODUCTS_BEFOR_PUSHER.LENGHT].IS_ACTUAL := TRUE;

   //Присвоение ID изделию
   "ITEMS_COLLECTION".PRODUCTS_BEFOR_PUSHER.PRODUCTS["ITEMS_COLLECTION".PRODUCTS_BEFOR_PUSHER.LENGHT].ID := "ITEMS_COLLECTION".PRODUCTS_BEFOR_PUSHER.INDEX;

   //Инкрементация счетчика изделий
   "ITEMS_COLLECTION".PRODUCTS_BEFOR_PUSHER.INDEX := "ITEMS_COLLECTION".PRODUCTS_BEFOR_PUSHER.INDEX + 1;

   //Добавление длины данных
   "ITEMS_COLLECTION".PRODUCTS_BEFOR_PUSHER.LENGHT := "ITEMS_COLLECTION".PRODUCTS_BEFOR_PUSHER.LENGHT + 1;
END_FUNCTION

FUNCTION "COMPARE_ID" : Bool   // FC7, LAD
TITLE = Сравнение GTIN
{ S7_Optimized_Access := 'TRUE' }
VERSION : 0.1
   VAR_INPUT
      ID_FROM_TASK : String;
      ID_FROM_SCAN_RESULT : String;
   END_VAR
   VAR_TEMP
      CHARS_FROM_TASK : Array[0..40] of Char;
      CHARS_FROM_TASK_LENGHT : Int;
      CHARS_FROM_SCAN_RESULT : Array[0..40] of Char;
      CHARS_FROM_SCAN_RESULT_LENGHT : Int;
      CONTER : Int;
   END_VAR
BEGIN

REGION Network 1 (SCL): Получение символов из ID задания
   Strg_TO_Chars(Strg:=#ID_FROM_TASK,
                 pChars:=0,
                 Cnt=>#CHARS_FROM_TASK_LENGHT,
                 Chars:=#CHARS_FROM_TASK);
END_REGION

REGION Network 2 (SCL): Получение символов из ID результата сканирования
   Strg_TO_Chars(Strg := #ID_FROM_SCAN_RESULT,
                 pChars := 0,
                 Cnt => #CHARS_FROM_SCAN_RESULT_LENGHT,
                 Chars := #CHARS_FROM_SCAN_RESULT);
END_REGION

REGION Network 3 (SCL): Сравнение длины строк
   // Если длина обеих строк не равна, возвращаем FALSE
   IF #CHARS_FROM_TASK_LENGHT <> #CHARS_FROM_SCAN_RESULT_LENGHT THEN

       //Устанавливаем результат выполнения функции
       #COMPARE_ID := FALSE;

       //Устанавливаем ошибке
       "ALARMS".ALARMS.ERROR_2_FS2_FAULT := TRUE;

       //Выход из функции
       RETURN;
   END_IF;
END_REGION

REGION Network 4 (SCL): Посимвольное сравнение строк
   FOR #CONTER := 0 TO #CHARS_FROM_TASK_LENGHT DO

       IF #CHARS_FROM_TASK[#CONTER] <> #CHARS_FROM_SCAN_RESULT[#CONTER] THEN

           //Устанавливаем результат выполнения функции
           #COMPARE_ID := FALSE;

           //Устанавливаем ошибке
           "ALARMS".ALARMS.ERROR_2_FS2_FAULT := TRUE;
           "ALARMS".ALARMS.ERROR_2_FS2_FAULT := TRUE;

           //Выход из функции
           RETURN;

       END_IF;

   END_FOR;
END_REGION

REGION Network 5 (SCL): Возврат результата сравнения TRUE
   // Если ранее из функции не вышли, значит строки одинаковые.
   //Устанавливаем результат выполнения функции
   #COMPARE_ID := TRUE;

   //Выход из функции
   RETURN;
END_REGION
END_FUNCTION

FUNCTION "WORD_TO_BYTES" : Void   // FC11, LAD
{ S7_Optimized_Access := 'TRUE' }
VERSION : 0.1
   VAR_INPUT
      IN_WORD : Word;
   END_VAR
   VAR_OUTPUT
      LO_BYTE : Byte;
      HI_BYTE : Byte;
   END_VAR
BEGIN

REGION Network 1 (SCL)
   "wBuffer" := #IN_WORD;
   #HI_BYTE := "HiChar";
   #LO_BYTE := "loChar";
END_REGION
END_FUNCTION

FUNCTION "UDINT_TO_STR" : Void   // FC14, LAD
{ S7_Optimized_Access := 'TRUE' }
VERSION : 0.1
   VAR_INPUT
      IN : UDInt;
   END_VAR
   VAR_OUTPUT
      OUT : String;
   END_VAR
BEGIN

REGION Network 1
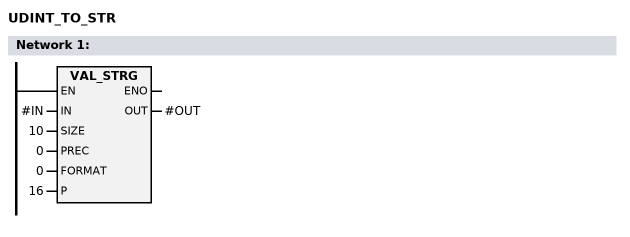
   VAL_STRG(IN := #IN, SIZE := 10, PREC := 0, FORMAT := 0, P := 16, OUT => #OUT);
END_REGION
END_FUNCTION

// folder: 1_MAIN_INTERLOCK

FUNCTION "INTERLOCK" : Void   // FC2, FBD
{ S7_Optimized_Access := 'TRUE' }
VERSION : 0.1
   VAR_INPUT
      UPS_OK : Bool;   // Сигнал от ИБП
   END_VAR
   VAR_TEMP
      buzzerActivate : Bool;
      ups_fault_delay : Bool;
   END_VAR
   VAR_TEMP   // added for the SCL form of the ladder/FBD networks
      _w1 : Bool;
   END_VAR
BEGIN

REGION Network 1: Формирование задержки для ошибки ИБП
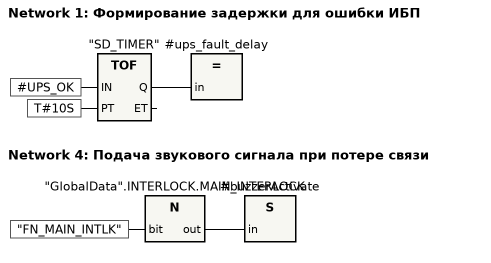
   "SD_TIMER".TOF(IN := #UPS_OK, PT := T#10S);
   #ups_fault_delay := "SD_TIMER".Q;
END_REGION

REGION Network 2 (SCL): Обработка ошибки питания от ИБП
   // При появлении ошибки питания от ИБП формируем сообщение об ошибке
   //Если поступил сигнал об ошибке от ИБП
   IF #ups_fault_delay = FALSE THEN
       "GlobalData".INTERLOCK.MAIN_INTERLOCK := FALSE;
       "GlobalData".FROM_HMI.CTW.RUN_CMD_FROM_HMI := FALSE;
       "ALARMS".ALARMS.ERROR_POWER_SYPLE := TRUE;
   END_IF;

   //Если сигнал об ошибке от ИБП пропал
   IF #UPS_OK = TRUE THEN
       "ALARMS".ALARMS.ERROR_POWER_SYPLE := FALSE;
   END_IF;
END_REGION

REGION Network 3 (SCL): Обработка разрыва связи с ПК
   // БЛОК ОТСЛЕЖИВАЕТ НАЛИЧИЕ КОММУНИКАЦИИ
   //     МЕЖДУ ПК И ПЛК. В СЛУЧАЕ ОТСУТСВИЯ КОММУНИКАЦИИ
   //     РАЗРЕШЕНИЕ НА РАБОТУ МЕХАНИЗМОВ БЛОКИРУЕТСЯ
   //     
   //     Каждый раз ПК сбрасывает счетчик времени между сессиями. 
   //     В прерывании OB30 инкрементируется счетчик времени между сессиями. 
   //     При достижении порогового значения устанавливается разрыв соединения
   (*
       ФУНКЦИЯ ОТСЛЕЖИВАЕТ НАЛИЧИЕ КОММУНИКАЦИИ
       МЕЖДУ ПК И ПЛК. В СЛУЧАЕ ОТСУТСВИЯ КОММУНИКАЦИИ
       РАЗРЕШЕНИЕ НА РАБОТУ МЕХАНИЗМОВ БЛОКИРУЕТСЯ

       Каждый раз ПК сбрасывает счетчик времени между сессиями. 
       В прерывании OB30 инкрементируется счетчик времени между сессиями. 
       При достижении порогового значения устанавливается разрыв соединения
   *)

   // Если счетчик превысил значение, сбрасываем команду
   // для работы установки (50 х 100 мсек = 5 сек)
   IF "GlobalData".INTERLOCK.DISCONNECT_COUNTER > 50 THEN
       "GlobalData".INTERLOCK.MAIN_INTERLOCK := FALSE;
   END_IF;

   //Если появилась команда для сброса счеткика - сбрасываем его
   IF "GlobalData".INTERLOCK.RESET_COUNTER_DISCONNECT = TRUE THEN
       "GlobalData".INTERLOCK.RESET_COUNTER_DISCONNECT := FALSE;
       "GlobalData".INTERLOCK.MAIN_INTERLOCK := TRUE;
       "GlobalData".INTERLOCK.DISCONNECT_COUNTER := 0;
   END_IF;

   //Если главная деблокировка пропала, сбрасываем команду
   //на работу межанизмов
   IF "GlobalData".INTERLOCK.MAIN_INTERLOCK = FALSE THEN
       "GlobalData".FROM_HMI.CTW.RUN_CMD_FROM_HMI := FALSE;
       "GlobalData".FROM_HMI.CTW.CONVEYOR_FORCE_RUN := FALSE;
   END_IF;
END_REGION

REGION Network 4: Подача звукового сигнала при потере связи
   #_w1 := NOT "GlobalData".INTERLOCK.MAIN_INTERLOCK AND "FN_MAIN_INTLK";   // falling edge of "GlobalData".INTERLOCK.MAIN_INTERLOCK
   "FN_MAIN_INTLK" := "GlobalData".INTERLOCK.MAIN_INTERLOCK;
   IF #_w1 THEN #buzzerActivate := TRUE; END_IF;
END_REGION

REGION Network 5 (SCL)
   IF "GlobalData".FROM_HMI.CTW.HMI_IS_RUN = TRUE AND #buzzerActivate = TRUE THEN
       "GlobalData".AUX.BUZZER_ACTIVATE := TRUE;
   END_IF;
END_REGION
END_FUNCTION

// folder: 2_КОНВЕЙЕР

FUNCTION_BLOCK "CONVEYOR"   // FB2, LAD
{ S7_Optimized_Access := 'TRUE' }
VERSION : 0.1
   VAR_INPUT
      RUN_IN : Bool;   // Сигнал для запуска конвейера
      FORCE_RUN : Bool;   // Сигнал для принудительного запуска конвейера
   END_VAR
   VAR_OUTPUT
      RUN_OUT : Bool;   // Выход на пускатель конвейера
      GREEN_LAMP : Bool;   // Зеленая лампа световой сигнализации
      RED_LAMP : Bool;   // Красная лампа световой сигнализации
      LINE_IS_RUN_NORMAL_MODE : Bool;   // Линия работает в нормальном режиме
   END_VAR
   VAR
      IEC_Timer_0_Instance : TON_TIME;
   END_VAR
   VAR_TEMP
      StartNormalRequest : Bool;   // Запрос для включения конвейера в нормальном режиме
      StartForceRequest : Bool;   // Запрос на включение конвейера в принудительном режиме
   END_VAR
BEGIN

REGION Network 1: Запрос на включение конвейера в нормальном режиме
   // Запуск конвейера в нормальном режиме может быть осуществлен при следующих условиях:
   // 1. Подан сигнал на включение конвейера в нормальном режиме
   // 2. Отсутсвует запрос на включение конвейера в принудительном режиме
   // 3. Отсутствуют ошибки, препятствующие запуску конвейера
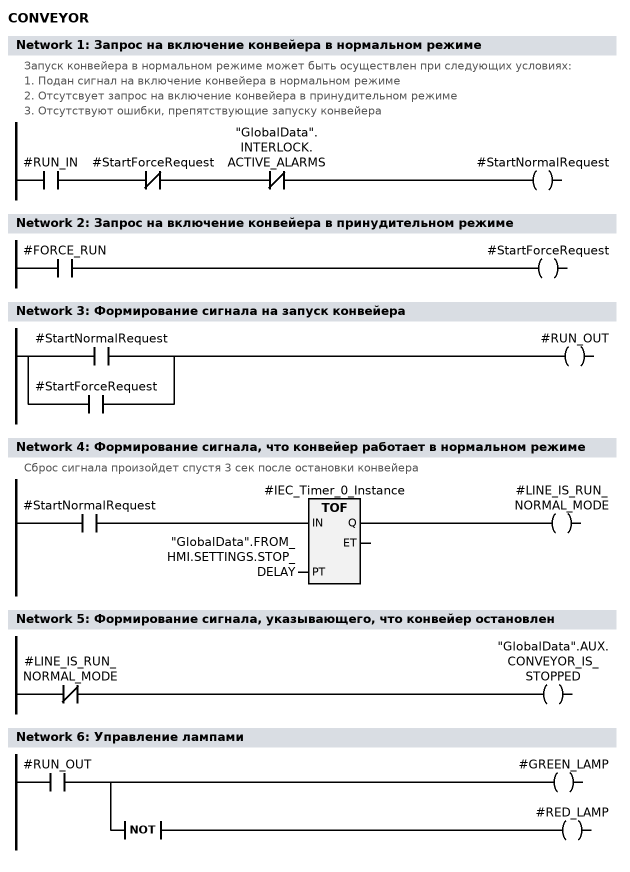
   RUNG wire#powerrail
      Contact( #RUN_IN )
      I_Contact( #StartForceRequest )
      I_Contact( "GlobalData".INTERLOCK.ACTIVE_ALARMS )
      Coil( #StartNormalRequest )
   END_RUNG
   // the same network as SCL:
   #StartNormalRequest := #RUN_IN AND NOT #StartForceRequest AND NOT "GlobalData".INTERLOCK.ACTIVE_ALARMS;
END_REGION

REGION Network 2: Запрос на включение конвейера в принудительном режиме
   RUNG wire#powerrail
      Contact( #FORCE_RUN )
      Coil( #StartForceRequest )
   END_RUNG
   // the same network as SCL:
   #StartForceRequest := #FORCE_RUN;
END_REGION

REGION Network 3: Формирование сигнала на запуск конвейера
   RUNG wire#powerrail
      Contact( #StartNormalRequest )
      wire#w1
      Coil( #RUN_OUT )
   END_RUNG
   RUNG wire#powerrail
      Contact( #StartForceRequest )
   END_RUNG wire#w1
   // the same network as SCL:
   #RUN_OUT := #StartNormalRequest OR #StartForceRequest;
END_REGION

REGION Network 4: Формирование сигнала, что конвейер работает в нормальном режиме
   // Сброс сигнала произойдет спустя 3 сек после остановки конвейера
   #IEC_Timer_0_Instance(IN := #StartNormalRequest, PT := "GlobalData".FROM_HMI.SETTINGS.STOP_DELAY);   // TOF
   #LINE_IS_RUN_NORMAL_MODE := #IEC_Timer_0_Instance.Q;
END_REGION

REGION Network 5: Формирование сигнала, указывающего, что конвейер остановлен
   RUNG wire#powerrail
      I_Contact( #LINE_IS_RUN_NORMAL_MODE )
      Coil( "GlobalData".AUX.CONVEYOR_IS_STOPPED )
   END_RUNG
   // the same network as SCL:
   "GlobalData".AUX.CONVEYOR_IS_STOPPED := NOT #LINE_IS_RUN_NORMAL_MODE;
END_REGION

REGION Network 6: Управление лампами
   RUNG wire#powerrail
      Contact( #RUN_OUT )
      wire#w1
      Coil( #GREEN_LAMP )
   END_RUNG
   RUNG wire#w1
      Not()
      Coil( #RED_LAMP )
   END_RUNG
   // the same network as SCL:
   #GREEN_LAMP := #RUN_OUT;
   #RED_LAMP := NOT #RUN_OUT;
END_REGION
END_FUNCTION_BLOCK

// folder: 4_СКАНЕР MATRIX

FUNCTION_BLOCK "mSCANER"   // FB13, LAD
TITLE = СКАНЕР
{ S7_Optimized_Access := 'FALSE' }
VERSION : 0.1
// Блок управляет работой сканера
   VAR_INPUT
      INTERLOCK : Bool;   // Деблокировка для работы сканера
      FS1 : Bool;   // Состояние фотодатчика
      GOOD_READ : Bool;   // Сигнал об сканера о том, что код считался
      NO_READ : Bool;   // Сигнал от сканера, что код не считался
   END_VAR
   VAR_OUTPUT
      PHASE_ON : Bool;   // Сигнал для начала фазы сканирования
      PHASE_OFF : Bool;   // Сигнал для завершения фазы сканирования
      STAGE : UInt;   // Этап, на котором находится выполнение блока
   END_VAR
   VAR
      cycleStart : DTL;   // Время, при котором начат цикл
      FS1_OLDSTATE : Bool;   // Предыдущее значение фотодатчика сканера
      oldGoodRead : Bool;
      oldNoRead : Bool;
      goodReadMemmoryFlag : Bool;
      noReadMemmoryFlag : Bool;
      busy : Bool;
      ProductsAreTooCloseToEachOther : Bool;   // Продукты слишком близко друг к другу
   END_VAR
   VAR_TEMP
      Status : Word;
      FS_FRONT_POSITIVE : Bool;   // Передний фронт сигнала фотодатчика
      currentTime : DTL;   // Текущее время
      timeDelta : Time;   // Дельта времени (вычисляется каждый раз)
      tmpResult : Int;
      emptyData : Bool;
      gtinIsEquals : Bool;   // Флаг, указывающий, что GTIN задания и результата сканирования совпадают
      barcodeIsEquals : Bool;   // Флаг, указывающий, что штрихкод задания и результата сканирования совпадают
      Index : UDInt;
      i : Int;
      symbolH : Char;
      symbolL : Char;
      dataProcessing : Bool;   // Фдаг для обработки данных, полученных от сканера
   END_VAR
BEGIN

REGION Network 1 (SCL): ОБРАБОТКА ОТСУТСТВИЯ ДЕБЛОКИРОВКИ
   // В случае отсутсвия деблокировки сбрасываем все переменные и выключаем сканер
   IF #INTERLOCK = FALSE THEN

       //Устанавливаем этап выполнения блока
       #STAGE := 0;

       //Выключаем сканер
       #PHASE_ON := FALSE;
       #PHASE_OFF := FALSE;

       //Выходим из функции
       RETURN;

   END_IF;
END_REGION

REGION Network 2 (SCL): ВЫДЕЛЕНИЕ ПОЛОЖИТЕЛЬНОГО ФРОНТА СИГНАЛА ФОТОДАТЧИКА FS1
   #FS_FRONT_POSITIVE := #FS1 = TRUE AND #FS1_OLDSTATE = FALSE;
   #FS1_OLDSTATE := #FS1;
END_REGION

REGION Network 3 (SCL): ФОРМИРОВАНИЕ ОШИБКИ - ПРОДУКТ СЛИШКОМ БЛИЗКО
   //Если модуль сканирования не завершил работу и на входе появился
   //продукт - устанавливаем ошибку
   IF #FS_FRONT_POSITIVE = TRUE AND #busy = TRUE THEN

       #ProductsAreTooCloseToEachOther := TRUE;

   END_IF;
END_REGION

REGION Network 4 (SCL): ОБРАБОТКА ПОЛОЖИТЕЛЬНОГО ФРОНТА СИГНАЛА ФОТОДАТЧИКА 1
   // При срабатывании фотодатчика 1 устанавливаем флаг, что возник передний фронт
   // Устанавливаем фазу работы блока: 1
   // Добавляем новое изделие в колекцию изделий между сканером и отбраковщиком
   //Установка фазы работы блока
   IF #FS_FRONT_POSITIVE = TRUE AND #busy = FALSE THEN

       //Установка статуса - этап 1 (начало ожидания
       //для включения сканера)
       #STAGE := 1;

       //Получаем системное время при котором
       //выход фотодатчика изменил свое состояние
       #tmpResult := RD_SYS_T(OUT => #cycleStart);

       //Устанавливаем флаг, что приложение занято
       #busy := TRUE;

   END_IF;
END_REGION

REGION Network 5 (SCL): ВЫХОД ИЗ БЛОКА ПРИ ОТСУТСТВИИ ЗАДАЧИ
   // В случае, если не выполняется ни одна фаза работы блока, покидаем функцию
   IF #STAGE = 0 THEN

       //Сброс вспомогательных значений
       #goodReadMemmoryFlag := FALSE;
       #noReadMemmoryFlag := FALSE;

       #busy := FALSE;

       RETURN;

   END_IF;
END_REGION

REGION Network 6 (SCL): ВЫЧИСЛЕНИЕ ТЕКУЩЕГО ВРЕМЕНИ
   //Запоминаем текущее время
   #tmpResult := RD_SYS_T(OUT => #currentTime);

   //Вычисление времени с начала цикла
   #timeDelta := #currentTime - #cycleStart;
END_REGION

REGION Network 7 (SCL): ФАЗА 1 - ВКЛЮЧЕНИЕ СКАНЕРА
   IF #STAGE = 1 AND (#timeDelta > "GlobalData".FROM_HMI.SETTINGS.TIME_A) THEN

       //Очистка буфера от старых значений
       FOR #i := 0 TO 100 DO
           "MODBUS_DATA".MODBUS_DATA[#i] := 0;
       END_FOR;

       //Установка состояний выходных сигналов
       #PHASE_ON := TRUE;
       #PHASE_OFF := FALSE;

       //Установка статуса - этап 2 (включение сканера)
       #STAGE := 2;

   END_IF;
END_REGION

REGION Network 8 (SCL): ФАЗА 2 - ВЫКЛЮЧЕНИЕ СКАНЕРА ПО ИСТЕЧЕНИЮ ВРЕМЕНИ
   IF ((#timeDelta >= ("GlobalData".FROM_HMI.SETTINGS.TIME_A + "GlobalData".FROM_HMI.SETTINGS.TIME_B))  AND #STAGE = 2) THEN

       #PHASE_ON := FALSE;
       #PHASE_OFF := FALSE;

       //Установка статуса - этап 3 (выключение сканера)
       #STAGE := 3;

   END_IF;
END_REGION

REGION Network 9 (SCL): ОБРАБОТКА СИГНАЛОВ GOOD_READ и NO_READ
   // Если на этапе сканирования появились сигналы  #GOOD_READ или #NO_READ - запоминаем это
       IF (#GOOD_READ = TRUE AND #oldGoodRead = FALSE AND #STAGE >= 2) THEN
           #goodReadMemmoryFlag := TRUE;
       END_IF;

       IF (#NO_READ = TRUE AND #oldNoRead = FALSE AND #STAGE = 2) THEN
           #noReadMemmoryFlag := TRUE;
       END_IF;

   #oldGoodRead := #GOOD_READ;
   #oldNoRead := #NO_READ;
END_REGION

REGION Network 10 (SCL): ФАЗА 3- ЗАВЕРШЕНИЕ ОЖИДАНИЯ РЕЗУЛЬТАТА СКАНИРОВАНИЯ ПО ТАЙМАУТУ
   IF ((#timeDelta >= ("GlobalData".FROM_HMI.SETTINGS.TIME_A + "GlobalData".FROM_HMI.SETTINGS.TIME_C) AND #STAGE = 3)) THEN

       //Установка состояний выходных сигналов
       #PHASE_ON := FALSE;
       #PHASE_OFF := TRUE;

       //Установка флага, для того, чтоб данные
       //полученые из сканера обработались
       #dataProcessing := TRUE;

   END_IF;
END_REGION

REGION Network 11 (SCL): Установка флагов для обработки принятых данных
       //Если стадия выполнения блока 2 (сканирование)
       //тогда обрабатываем сигналы #GOOD_READ и #NO_READ
       IF (#dataProcessing = TRUE) THEN

           //Сброс флага для того, чтоб данные обрабатывались 
           //только один раз при взводе флага
           #dataProcessing := FALSE;

           // В тестовом режиме искуственно устанавливаем флаг GOOD_REED и сбрасываем NO_READ

           IF ("TestMode" = TRUE) THEN
               #goodReadMemmoryFlag := TRUE;
               #noReadMemmoryFlag := FALSE;
           END_IF;


           //Определение положительного фронта для сигнала GOOD_READ
           IF (#goodReadMemmoryFlag = TRUE) THEN

               #goodReadMemmoryFlag := FALSE;

               #PHASE_ON := FALSE;
               #PHASE_OFF := TRUE;

               //Перемещение кода
               //Получаем текущий индекс в коллекции
               #Index := "ITEMS_COLLECTION".PRODUCTS_BEFOR_PUSHER.LENGHT;


               // В рабочем режиме перенос данных из Modbus в поле продукта            
               IF ("TestMode" = FALSE) THEN

                   "MODBUS_DATA_TO STRING"("ITEMS_COLLECTION".PRODUCTS_BEFOR_PUSHER.PRODUCTS[#Index].BARCODE);
               END_IF;

               // В тестовом режиме запуск функции чтения кодов из тестовой базы данных и перенос в поле продукта
               IF ("TestMode" = TRUE) THEN

                   "TestCodesGenerate_DB"("TestDB".Index_for_testproduct);
                   "ITEMS_COLLECTION".PRODUCTS_BEFOR_PUSHER.PRODUCTS[#Index].BARCODE := "TestDB".Actual_testproduct;
                   "ITEMS_COLLECTION".PRODUCTS_BEFOR_PUSHER.PRODUCTS[#Index].IS_GOOD := TRUE;


               END_IF;


               //Если штрихкод не пустой
               IF "ITEMS_COLLECTION".PRODUCTS_BEFOR_PUSHER.PRODUCTS[#Index].BARCODE <> '' THEN

                   "ITEMS_COLLECTION".PRODUCTS_BEFOR_PUSHER.PRODUCTS[#Index].IS_GOOD := TRUE;

               END_IF;

               //Передача прочих свойств продукту
               "ITEMS_COLLECTION".PRODUCTS_BEFOR_PUSHER.PRODUCTS[#Index].IS_ACTUAL := TRUE;
               "ITEMS_COLLECTION".PRODUCTS_BEFOR_PUSHER.PRODUCTS[#Index].ID := "ITEMS_COLLECTION".PRODUCTS_BEFOR_PUSHER.INDEX;

               //Помещение в блоке изделия, прошедщего отбраковщик
          //     "GlobalData".PRODUCT_IS_SCANING_AREA := "ITEMS_COLLECTION".PRODUCTS_BEFOR_PUSHER.PRODUCTS[#Index];

               //Инкрементация счетчикацц
               "ITEMS_COLLECTION".PRODUCTS_BEFOR_PUSHER.LENGHT := "ITEMS_COLLECTION".PRODUCTS_BEFOR_PUSHER.LENGHT + 1;
               "ITEMS_COLLECTION".PRODUCTS_BEFOR_PUSHER.INDEX := "ITEMS_COLLECTION".PRODUCTS_BEFOR_PUSHER.INDEX + 1;

               //Установка этапа выполнения блока
               #STAGE := 0;

               //Выход из функции
               RETURN;

           END_IF;

           ///Определение положительного фронта для сигнала NO_READ
           //IF (#noReadMemmoryFlag = TRUE) THEN

               #noReadMemmoryFlag := FALSE;

               #PHASE_ON := FALSE;
               #PHASE_OFF := TRUE;

               //Перемещение кода
               //Получаем текущий индекс в коллекции
               #Index := "ITEMS_COLLECTION".PRODUCTS_BEFOR_PUSHER.LENGHT;

               //Передача свойств изделию
               "ITEMS_COLLECTION".PRODUCTS_BEFOR_PUSHER.PRODUCTS[#Index].IS_ACTUAL := TRUE;
               "ITEMS_COLLECTION".PRODUCTS_BEFOR_PUSHER.PRODUCTS[#Index].IS_GOOD := FALSE;

               //Очистка кода
               //Перенос данных из буфера сканера
               //в экземпляр продукта
               "ITEMS_COLLECTION".PRODUCTS_BEFOR_PUSHER.PRODUCTS[#Index].BARCODE := '';

               //Инкрементация счетчика
               "ITEMS_COLLECTION".PRODUCTS_BEFOR_PUSHER.LENGHT := "ITEMS_COLLECTION".PRODUCTS_BEFOR_PUSHER.LENGHT + 1;
               "ITEMS_COLLECTION".PRODUCTS_BEFOR_PUSHER.INDEX := "ITEMS_COLLECTION".PRODUCTS_BEFOR_PUSHER.INDEX + 1;

               //Установка этапа выполнения блока
               #STAGE := 0;

          // END_IF;
       END_IF;
END_REGION
END_FUNCTION_BLOCK

FUNCTION "MODBUS_TCP_MASTER" : Void   // FC9, FBD
{ S7_Optimized_Access := 'TRUE' }
VERSION : 0.1
   VAR_TEMP
      NDR : Bool;
      DR : Bool;
      ERROR : Bool;
      STATUS : Word;
   END_VAR
BEGIN

REGION Network 1
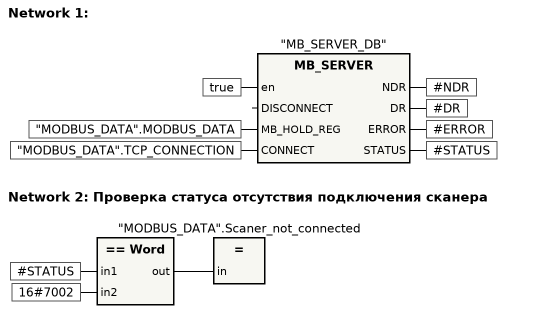
   IF true THEN
       "MB_SERVER_DB"(MB_HOLD_REG := "MODBUS_DATA".MODBUS_DATA,   // MB_SERVER
                      CONNECT := "MODBUS_DATA".TCP_CONNECTION,
                      NDR => #NDR,
                      DR => #DR,
                      ERROR => #ERROR,
                      STATUS => #STATUS);
   END_IF;
END_REGION

REGION Network 2: Проверка статуса отсутствия подключения сканера
   "MODBUS_DATA".Scaner_not_connected := #STATUS = 16#7002;
END_REGION
END_FUNCTION

FUNCTION "MODBUS_DATA_TO STRING" : Void   // FC12, LAD
{ S7_Optimized_Access := 'TRUE' }
VERSION : 0.1
   VAR_IN_OUT
      InOut_Str : String;
   END_VAR
   VAR_TEMP
      i : DInt;
      _byte : Byte;
   END_VAR
BEGIN

REGION Network 1 (SCL)

       //Копирование данных из одной области памяти
       //в другую
       FOR #i := 0 TO 200 DO

           #_byte := PEEK(area := 16#84,
                          dbNumber := 9,
                          byteOffset := 14 + #i);

           POKE(area := 16#84,
                dbNumber := 9,
                byteOffset := 216 + #i,
                value := #_byte);

       END_FOR;


       //Перенос данных из буфера сканера
       ////в выходную строку
       Chars_TO_Strg(Chars := "MODBUS_DATA".BYTES_ARRAY,
                     pChars := 0,
                     Cnt := 0,
                     Strg => #InOut_Str);
END_REGION
END_FUNCTION

// folder: 5_ОТБРАКОВЩИК

FUNCTION_BLOCK "PUSHER_CONTROL"   // FB1, LAD
TITLE = Блок, осуществляющий проверку работы отбраковщика
{ S7_Optimized_Access := 'TRUE' }
VERSION : 0.1
   VAR_INPUT
      INTERLOCK : Bool;   // Деблокировка для работы блока
      RESET : Bool;   // Команда для сброса блока
      FS3 : Bool;   // Состояние фотодатчика после отбраковщика
   END_VAR
   VAR_OUTPUT
      STAGE : Int;
   END_VAR
   VAR
      cycleStart : DTL;   // Время, при котором начат цикл
      FS3_OLDSTATE : Bool;   // Состояние фотодатчика в прошлос цикле
      FS3_ISSET : Bool;   // Переменая для сохранения состояния фотодатчика FS2
      busy : Bool;
   END_VAR
   VAR_TEMP
      FS_FRONT_POSITIVE : Bool;   // Положительный фронт фотодатчика
      tmpResult : Int;
      index : Int;   // Индекс для работы вцикле
      currentItem : "PRODUCT";   // Изделие, ближайшее к толкателю
      currentTime : DTL;   // Текущее время
      timeDelta : Time;   // Дельта времени (вычисляется каждый раз)
      PushDelayTime : Time;   // Время задержки срабатывания толкателя
      PushImpulsTime : Time;   // Время импульса
      PushCheckTime : Time;   // Время контроля отбраковки
   END_VAR
   VAR_TEMP   // added for the SCL form of the ladder/FBD networks
      _w1 : Bool;
   END_VAR
BEGIN

REGION Network 1 (SCL): ОБРАБОТКА ОТСУТСТВИЯ ДЕБЛОКИРОВКИ
   // В случае отсутсвия деблокировки сбрасываем все переменные
   IF #INTERLOCK = FALSE THEN

       #FS3_ISSET := FALSE;
       "Control_begin" := FALSE;
       #STAGE:=0;
       //Выходим из функции
       RETURN;

   END_IF;
END_REGION

REGION Network 2: Если появился флаг на запуск контроля отбраковки начинаем этот процесс
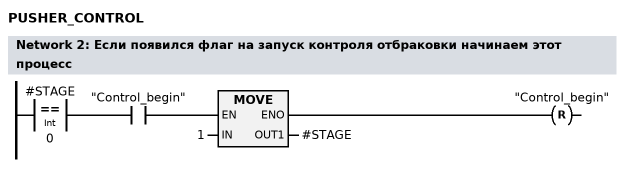
   RUNG wire#powerrail
      { S7_Templates := "SrcType := Int" } EQ_Contact(in1 := #STAGE, in2 := 0)
      Contact( "Control_begin" )
      Move(in := 1, out1 => #STAGE)
      R_Coil( "Control_begin" )
   END_RUNG
   // the same network as SCL:
   #_w1 := (#STAGE = 0) AND "Control_begin";
   IF #_w1 THEN
       #STAGE := 1;
       "Control_begin" := FALSE;
   END_IF;
END_REGION

REGION Network 3 (SCL): Запоминаем время начала цикла контроля отбраковки
   IF #STAGE = 1 THEN
       #tmpResult := RD_SYS_T(OUT => #cycleStart);
       #STAGE := 2;
   END_IF;
END_REGION

REGION Network 4 (SCL): ВЫДЕЛЕНИЕ ПОЛОЖИТЕЛЬНОГО ФРОНТА СИГНАЛА FS3
   #FS_FRONT_POSITIVE := #FS3 = TRUE AND #FS3_OLDSTATE = FALSE;
   #FS3_OLDSTATE := #FS3;
END_REGION

REGION Network 5 (SCL): ОБРАБОТКА ПОЛОЖИТЕЛЬНОГО ФРОНТА СИГНАЛА от датчика 3, когда идет процесс контроля отбраковки
   (*
       ПРОЦЕДУРА ВЫПОЛНЯЕТСЯ ПРИ СМЕНЕ СОСТОЯНИЯ 
       ВЫХОДА ФОТОДАТЧИКА НА TRUE
   *)
   IF #FS_FRONT_POSITIVE = TRUE AND #STAGE >= 2 THEN

       //Cообщаем об
       //необходимости ручной отбраковки
       "ALARMS".ALARMS.ERROR_6_ERROR_PUSHER := TRUE;

   END_IF;
END_REGION

REGION Network 6 (SCL): ПОДГОТОВКА ПЕРЕМЕННЫХ
   //Запоминаем текущее время
   #tmpResult := RD_SYS_T(OUT => #currentTime);

   //Вычисление времени с начала цикла
   #timeDelta := #currentTime - #cycleStart;

   //Перенос данных из датаблока
   #PushCheckTime := "GlobalData".FROM_HMI.SETTINGS.TIME_E;
END_REGION

REGION Network 7 (SCL): Подсчет времени контроля обработки
   // Если время контроля истекло, то сбрасываем флаг
   IF ((#timeDelta >= #PushCheckTime) AND #STAGE >= 2) THEN

       #STAGE := 0;

   //К количеству изделий, прошедших через
   //отбраковщик добавляем еще одно
   "GlobalData".AUX.COUNTERS.QUANTITY_PRODUCTS_AUTO_REJECTED := "GlobalData".AUX.COUNTERS.QUANTITY_PRODUCTS_AUTO_REJECTED + 1;

   END_IF;
END_REGION
END_FUNCTION_BLOCK

FUNCTION_BLOCK "PUSHER"   // FB6, LAD
{ S7_Optimized_Access := 'TRUE' }
VERSION : 0.1
   VAR_INPUT
      INTERLOCK : Bool;   // Деблокировка для работы блока
      RESET : Bool;   // Команда для сброса блока
      FS2 : Bool;   // Состояние фотодатчика перед отбраковщиком
      FS3 : Bool;   // Состояние фотодатчика после отбраковщика
   END_VAR
   VAR_OUTPUT
      PUSHER_OUT : Bool;   // Выход толкателя
      STAGE : Int;
   END_VAR
   VAR
      cycleStart : DTL;   // Время, при котором начат цикл
      MassMarriageCounter : Int := 0;   // Счетчик массового брака
      FS2_OLDSTATE : Bool;   // Состояние фотодатчика в прошлос цикле
      FS2_ISSET : Bool;   // Переменая для сохранения состояния фотодатчика FS2
      ProductsAreTooCloseToEachOther : Bool;   // Продукты слишком близко друг к другу
      busy : Bool;
      "counter" : Int;
   END_VAR
   VAR_TEMP
      FS_FRONT_POSITIVE : Bool;   // Положительный фронт фотодатчика
      tmpResult : Int;
      index : UDInt;   // Индекс для работы вцикле
      currentIProduct : "PRODUCT";   // Изделие, ближайшее к толкателю
      currentTime : DTL;   // Текущее время
      timeDelta : Time;   // Дельта времени (вычисляется каждый раз)
      PushDelayTime : Time;   // Время задержки срабатывания толкателя
      PushImpulsTime : Time;   // Время импульса
      PushCheckTime : Time;   // Время контроля отбраковки
   END_VAR
BEGIN

REGION Network 1 (SCL): ОБРАБОТКА ОТСУТСТВИЯ ДЕБЛОКИРОВКИ
   // В случае отсутсвия деблокировки сбрасываем все переменные и выключаем толкатель отбраковщика
   IF #INTERLOCK = FALSE THEN

       //Устанавливаем этап выполнения блока
       #STAGE := 0;

       #FS2_ISSET := FALSE;

       //Выключаем толкатель
      //#PUSHER_OUT := FALSE;

       //Выходим из функции
       RETURN;

   END_IF;
END_REGION

REGION Network 2 (SCL): ВЫДЕЛЕНИЕ ПОЛОЖИТЕЛЬНОГО ФРОНТА СИГНАЛА ФОТОДАТ
   #FS_FRONT_POSITIVE := #FS2 = TRUE AND #FS2_OLDSTATE = FALSE;
   #FS2_OLDSTATE := #FS2;
END_REGION

REGION Network 3 (SCL): ФОРМИРОВАНИЕ ОШИБКИ - ПРОДУКТ СЛИШКОМ БЛИЗКО
   //Если отбраковщик не завершил работу и на входе появился
   //продукт - устанавливаем ошибку
   IF #FS_FRONT_POSITIVE = TRUE AND #busy = TRUE THEN

      #ProductsAreTooCloseToEachOther := TRUE;

   END_IF;
END_REGION

REGION Network 4 (SCL): ОБРАБОТКА ПОЛОЖИТЕЛЬНОГО ФРОНТА СИГНАЛА С ВЫХОДА ФОТОДАТЧИКА

   (*
       ПРОЦЕДУРА ВЫПОЛНЯЕТСЯ ПРИ СМЕНЕ СОСТОЯНИЯ 
       ВЫХОДА ФОТОДАТЧИКА НА TRUE
   *)
   IF #FS_FRONT_POSITIVE = TRUE AND #busy = FALSE THEN

       //Указываем, что блок занят выполнением 
       //задачи
       #busy := TRUE;

       //Получаем системное время при котором
       //выход фотодатчика изменил свое состояние
       #tmpResult := RD_SYS_T(OUT => #cycleStart);

       //Устанавливаем состояние выхода
       //толкателя как неактивно
      // #PUSHER_OUT := false;

       //Запоминаем изделие, находящееся ближе всего
       //к толкателю
       #currentIProduct := "ITEMS_COLLECTION".PRODUCTS_BEFOR_PUSHER.PRODUCTS[0];

       //Если изделие, ближайшее к толкателю не подлежит
       //отбраковке, устаналиваем флаг для считывания изделия
       IF #currentIProduct.IS_GOOD = TRUE THEN

         //Если штрихкод не пустая строка
           IF (#currentIProduct.BARCODE <> '') THEN

               //Получение индекса следующего продукта
               #index := "ITEMS_COLLECTION".PRODUCTS_IN_SEND_TO_PC.LENGHT;

               //Переносим продукта в коллекцию на отправку
               "ITEMS_COLLECTION".PRODUCTS_IN_SEND_TO_PC.PRODUCTS[#index] := #currentIProduct;

               //Обновление счетчика продуктов, подлежащих отправке
               "ITEMS_COLLECTION".PRODUCTS_IN_SEND_TO_PC.LENGHT := "ITEMS_COLLECTION".PRODUCTS_IN_SEND_TO_PC.LENGHT + 1;

               //Инкремент счетчика тестовой отправки
               "TestDB".counter_transfer_products := "TestDB".counter_transfer_products + 1;

          END_IF;

      END_IF;



       //Если изделие, ближайшее к толкателю подлежит
       //отбраковке, устаналиваем для этого соответсвующие переменные
       IF #currentIProduct.IS_GOOD = FALSE THEN
           #STAGE := 1;
       END_IF;

       //Сброс счеткика подряд отбракованых
       //изделий
       IF #currentIProduct.IS_GOOD = TRUE THEN

           //Обнуление счетчика брака
           "GlobalData".AUX.COUNTERS.DEFECT_COUNTER := 0;

       END_IF;

       //Сдвигаем коллекцию изделий, находящихся
       //между сканером и отбраковщиком вверх
       "SHIFT_UP_ITEMS_COLLECTION"();

   END_IF;
END_REGION

REGION Network 5 (SCL): ВЫХОД ИЗ ФУНКЦИИ ПРИ ОТСУТСТВИИ ЗАДАЧ
   //Если текущий этап не предусматривает действий,
   //выходим из функции, устанавливая выход толкателя
   //в неактивное состояние
   IF #STAGE = 0 THEN

       //#PUSHER_OUT := false;

       //Устанавливаем флаг, указывающий на 
       //то, что блок свободен для выполнения 
       //следующей задачи
       #busy := FALSE;

       //Выход из функции
       RETURN;

   END_IF;
END_REGION

REGION Network 6 (SCL): ПОДГОТОВКА ПЕРЕМЕННЫХ
   //Запоминаем текущее время
   #tmpResult := RD_SYS_T(OUT => #currentTime);

   //Вычисление времени с начала цикла
   #timeDelta := #currentTime - #cycleStart;

   //Перенос данных из датаблока
   #PushDelayTime := "GlobalData".FROM_HMI.SETTINGS.TIME_D;
   #PushImpulsTime := "GlobalData".FROM_HMI.SETTINGS.TIME_PUSHER_ACTIVE;
   #PushCheckTime := "GlobalData".FROM_HMI.SETTINGS.TIME_E;
END_REGION

REGION Network 7 (SCL): ЭТАП 1 - АКТИВАЦИЯ ТОЛКАТЕЛЯ
   // Если требуется отбраковка - активируется толкатель после задержки
       //Если имеется сигнал на активацию толкателя и время с начала цикла
       //не превысило время задержки работы толкателя, устанавливаем состояние выхода
       //в АКТИВНО
       IF #timeDelta >= #PushDelayTime AND #STAGE = 1   THEN

           //#PUSHER_OUT := TRUE;
           "IO".OUTPUTS.Pusher := TRUE;

           //устанавливаем флаг начала работы функции задвигания толкателя
           //"Флаг начала работы толкателя" := TRUE;

           #STAGE := 0;

       END_IF;
END_REGION

REGION Network 8 (SCL): ЭТАП 2- ДЕАКТИВАЦИЯ ТОЛКАТЕЛЯ
   // IF ((#timeDelta >= (#PushDelayTime + #PushImpulsTime)) AND #STAGE = 2) THEN

   //     #PUSHER_OUT := false;

   //     //Инкрементируем счетчик брака
   //     "GlobalData".AUX.COUNTERS.DEFECT_COUNTER := "GlobalData".AUX.COUNTERS.DEFECT_COUNTER + 1;

   //     #STAGE := 0;

   //     //устанавливаем флаг для начала контроля отбраковки продукта;

   //     "Control_begin" := TRUE;

   // END_IF;
END_REGION
END_FUNCTION_BLOCK

// folder: 6_КОЛЛЕКЦИЯ ИЗДЕЛИЙ

FUNCTION "SHIFT_UP_ITEMS_COLLECTION" : Void   // FC6, SCL
{ S7_Optimized_Access := 'TRUE' }
VERSION : 0.1
   VAR_TEMP
      Index : UDInt;
      "Counter" : UDInt;
      Lenght : UDInt;
   END_VAR
BEGIN
   (*
       СДВИГ ВВЕРХ КОЛЛЕКЦИИ ИЗДЕЛИЙ,
       НОХОДЯЩИХСЯ МЕЖДУ СКАНЕРОМ И ОТБРАКОВЩИКОМ
   *)

   #Counter := 0;
   #Lenght := "ITEMS_COLLECTION".PRODUCTS_BEFOR_PUSHER.#LENGHT;

   //Стираем данные из самой верхней
   //ячейки
   "ITEMS_COLLECTION".PRODUCTS_BEFOR_PUSHER.PRODUCTS[0].IS_ACTUAL := FALSE;
   //"ITEMS_COLLECTION".ITEMS[0].BARCODE := '';
   "ITEMS_COLLECTION".PRODUCTS_BEFOR_PUSHER.PRODUCTS[0].IS_GOOD := FALSE;


   //Цикл, в котором переносятся активные 
   //данные
   FOR #Index := 1 TO #Lenght DO

       IF "ITEMS_COLLECTION".PRODUCTS_BEFOR_PUSHER.PRODUCTS[#Index].IS_ACTUAL = TRUE THEN

           //Перемещение данных из временной коллекции в постояную
           "ITEMS_COLLECTION".PRODUCTS_BEFOR_PUSHER.PRODUCTS[#Counter] := "ITEMS_COLLECTION".PRODUCTS_BEFOR_PUSHER.PRODUCTS[#Index];

           //Инкрементация счетчика
           #Counter := #Counter + 1;

           CONTINUE;

       END_IF;

   END_FOR;

   //Цикл в котором все оставшиеся данные затираются
   FOR #Index := #Counter TO 20 DO

       "ITEMS_COLLECTION".PRODUCTS_BEFOR_PUSHER.PRODUCTS[#Index].IS_ACTUAL := FALSE;
       "ITEMS_COLLECTION".PRODUCTS_BEFOR_PUSHER.PRODUCTS[#Index].BARCODE := '';
       "ITEMS_COLLECTION".PRODUCTS_BEFOR_PUSHER.PRODUCTS[#Index].ID := 0;
       "ITEMS_COLLECTION".PRODUCTS_BEFOR_PUSHER.PRODUCTS[#Index].IS_GOOD := FALSE;

   END_FOR;

   //Передача количества изделий
   "ITEMS_COLLECTION".PRODUCTS_BEFOR_PUSHER.LENGHT := #Counter;
END_FUNCTION

FUNCTION "ITEMS_CONTROL" : Void   // FC8, LAD
{ S7_Optimized_Access := 'TRUE' }
VERSION : 0.1
BEGIN

REGION Network 1 (SCL): Процедура для очистки коллекции очереди
   IF "GlobalData".FROM_HMI.CTW.CLER_COLLECTION_CMD = TRUE THEN

       //Очистка коллекции
       "CLEAR"();

       //Сброс флага по которому происходит очистка коллекции
       "GlobalData".FROM_HMI.CTW.CLER_COLLECTION_CMD := FALSE;
   END_IF;
END_REGION
END_FUNCTION

FUNCTION "CLEAR" : Void   // FC10, LAD
{ S7_Optimized_Access := 'TRUE' }
VERSION : 0.1
   VAR_TEMP
      "Counter" : Int;
   END_VAR
BEGIN

REGION Network 1 (SCL): Очистка изделий
   //Цикл, в котором очищаются 
   //данные в коллекции перед буфером
   FOR #Counter := 0 TO 20 DO

       "ITEMS_COLLECTION".PRODUCTS_BEFOR_PUSHER.PRODUCTS[#Counter].IS_ACTUAL := FALSE;
       "ITEMS_COLLECTION".PRODUCTS_BEFOR_PUSHER.PRODUCTS[#Counter].BARCODE := '';
       "ITEMS_COLLECTION".PRODUCTS_BEFOR_PUSHER.PRODUCTS[#Counter].IS_GOOD := FALSE;
       "ITEMS_COLLECTION".PRODUCTS_BEFOR_PUSHER.PRODUCTS[#Counter].ID := 0;

   END_FOR;

   "ITEMS_COLLECTION".PRODUCTS_BEFOR_PUSHER.LENGHT := 0;
   "ITEMS_COLLECTION".PRODUCTS_BEFOR_PUSHER.INDEX := 0;

   //Цикл, в котором очищаются данные в коллекции на отправку
   FOR #Counter := 0 TO 3 DO

       "ITEMS_COLLECTION".PRODUCTS_IN_SEND_TO_PC.PRODUCTS[#Counter].IS_ACTUAL := FALSE;
       "ITEMS_COLLECTION".PRODUCTS_IN_SEND_TO_PC.PRODUCTS[#Counter].BARCODE := '';
       "ITEMS_COLLECTION".PRODUCTS_IN_SEND_TO_PC.PRODUCTS[#Counter].IS_GOOD := FALSE;
       "ITEMS_COLLECTION".PRODUCTS_IN_SEND_TO_PC.PRODUCTS[#Counter].ID := 0;

   END_FOR;

   "ITEMS_COLLECTION".PRODUCTS_IN_SEND_TO_PC.LENGHT := 0;
   "ITEMS_COLLECTION".PRODUCTS_IN_SEND_TO_PC.INDEX := 0;
END_REGION
END_FUNCTION

// folder: 7_СООБЩЕНИЯ

FUNCTION "ALARMS_FC" : Void   // FC3, LAD
{ S7_Optimized_Access := 'TRUE' }
VERSION : 0.1
   VAR_INPUT
      LineRunNormal : Bool;
   END_VAR
BEGIN

REGION Network 1 (SCL): Сброс всех ошибок
   // Если в слове управления поступила команда на сброс всех ошибок - осуществляем сброс всех ошибок
   IF "GlobalData".FROM_HMI.CTW.RESET_ALARMS_CMD = TRUE THEN

       %DB6.DBW4 := 0;
       %DB6.DBW6 := 0;

       %DB6.DBW12 := 0;
       %DB6.DBW14 := 0;

       "GlobalData".FROM_HMI.CTW.RESET_ALARMS_CMD := FALSE;

   END_IF;
END_REGION

REGION Network 2 (SCL): Обработка ошибки - массовый брак
   (*
       ФОРМИРОВАНИЕ ОШИБКИ ПРИ ПРЕВЫШЕНИИ СЧЕТЧИКА БРАКА
   *)
   IF "GlobalData".AUX.COUNTERS.DEFECT_COUNTER >= "GlobalData".FROM_HMI.SETTINGS.PRODUCT_DEFFECT_SETPOINT AND  "GlobalData".FROM_HMI.CTW.AUX_RUN_CMD = TRUE THEN
       "ALARMS".ALARMS.ERROR_7_OVER_DEFECT_COUNTER := TRUE;
   END_IF;

   (*
       СБРОС ОШИБКИ ЕСЛИ СЧЕТЧИК БРАКА НЕ ДОСТИГ ПРЕДЕЛА
   *)
   IF "GlobalData".AUX.COUNTERS.DEFECT_COUNTER < "GlobalData".FROM_HMI.SETTINGS.PRODUCT_DEFFECT_SETPOINT THEN
       "ALARMS".ALARMS.ERROR_7_OVER_DEFECT_COUNTER := FALSE;
   END_IF;

   (*
       ЕСЛИ ИЗМЕНИЛОСЬ ЗНАЧЕНИЕ НАСТРОЙКИ - МАССОВЫЙ БРАК
       ОБНУЛЯЕМ СЧЕТЧИК БРАКА
   *)
   IF "MEMMORYCELL_PRODUCT_DEFFECT_SETPOINT" <> "GlobalData".FROM_HMI.SETTINGS.PRODUCT_DEFFECT_SETPOINT THEN
       "MEMMORYCELL_PRODUCT_DEFFECT_SETPOINT" := "GlobalData".FROM_HMI.SETTINGS.PRODUCT_DEFFECT_SETPOINT;
       "GlobalData".AUX.COUNTERS.DEFECT_COUNTER := 0;
   END_IF;
END_REGION

REGION Network 3: Формирование ошибки - продукт в зоне сканера слишком близко
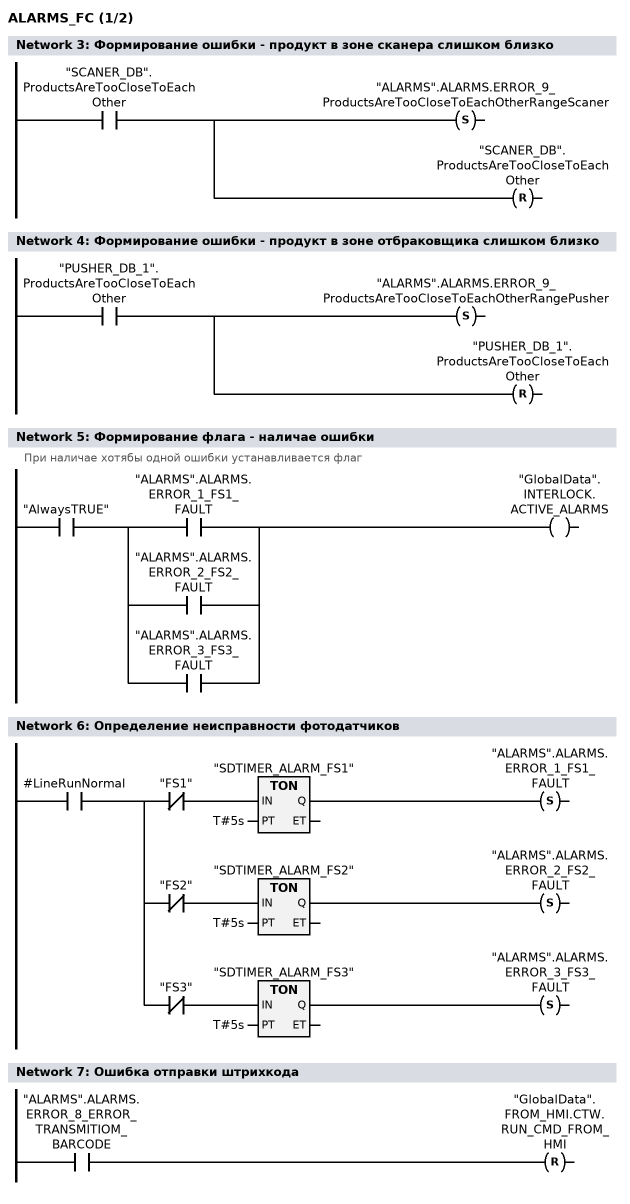
   RUNG wire#powerrail
      Contact( "SCANER_DB".ProductsAreTooCloseToEachOther )
      wire#w1
      S_Coil( "ALARMS".ALARMS.ERROR_9_ProductsAreTooCloseToEachOtherRangeScaner )
   END_RUNG
   RUNG wire#w1
      R_Coil( "SCANER_DB".ProductsAreTooCloseToEachOther )
   END_RUNG
   // the same network as SCL:
   IF "SCANER_DB".ProductsAreTooCloseToEachOther THEN
       "ALARMS".ALARMS.ERROR_9_ProductsAreTooCloseToEachOtherRangeScaner := TRUE;
       "SCANER_DB".ProductsAreTooCloseToEachOther := FALSE;
   END_IF;
END_REGION

REGION Network 4: Формирование ошибки - продукт в зоне отбраковщика слишком близко
   RUNG wire#powerrail
      Contact( "PUSHER_DB_1".ProductsAreTooCloseToEachOther )
      wire#w1
      S_Coil( "ALARMS".ALARMS.ERROR_9_ProductsAreTooCloseToEachOtherRangePusher )
   END_RUNG
   RUNG wire#w1
      R_Coil( "PUSHER_DB_1".ProductsAreTooCloseToEachOther )
   END_RUNG
   // the same network as SCL:
   IF "PUSHER_DB_1".ProductsAreTooCloseToEachOther THEN
       "ALARMS".ALARMS.ERROR_9_ProductsAreTooCloseToEachOtherRangePusher := TRUE;
       "PUSHER_DB_1".ProductsAreTooCloseToEachOther := FALSE;
   END_IF;
END_REGION

REGION Network 5: Формирование флага - наличае ошибки
   // При наличае хотябы одной ошибки устанавливается флаг
   RUNG wire#powerrail
      Contact( "AlwaysTRUE" )
      wire#w1
      Contact( "ALARMS".ALARMS.ERROR_1_FS1_FAULT )
      wire#w2
      Coil( "GlobalData".INTERLOCK.ACTIVE_ALARMS )
   END_RUNG
   RUNG wire#w1
      Contact( "ALARMS".ALARMS.ERROR_2_FS2_FAULT )
   END_RUNG wire#w2
   RUNG wire#w1
      Contact( "ALARMS".ALARMS.ERROR_3_FS3_FAULT )
   END_RUNG wire#w2
   // the same network as SCL:
   "GlobalData".INTERLOCK.ACTIVE_ALARMS := "AlwaysTRUE" AND ("ALARMS".ALARMS.ERROR_1_FS1_FAULT OR "ALARMS".ALARMS.ERROR_2_FS2_FAULT OR "ALARMS".ALARMS.ERROR_3_FS3_FAULT);
END_REGION

REGION Network 6: Определение неисправности фотодатчиков
   "SDTIMER_ALARM_FS1".TON(IN := #LineRunNormal AND NOT "FS1", PT := T#5s);
   IF "SDTIMER_ALARM_FS1".Q THEN "ALARMS".ALARMS.ERROR_1_FS1_FAULT := TRUE; END_IF;
   "SDTIMER_ALARM_FS2".TON(IN := #LineRunNormal AND NOT "FS2", PT := T#5s);
   IF "SDTIMER_ALARM_FS2".Q THEN "ALARMS".ALARMS.ERROR_2_FS2_FAULT := TRUE; END_IF;
   "SDTIMER_ALARM_FS3".TON(IN := #LineRunNormal AND NOT "FS3", PT := T#5s);
   IF "SDTIMER_ALARM_FS3".Q THEN "ALARMS".ALARMS.ERROR_3_FS3_FAULT := TRUE; END_IF;
END_REGION

REGION Network 7: Ошибка отправки штрихкода
   RUNG wire#powerrail
      Contact( "ALARMS".ALARMS.ERROR_8_ERROR_TRANSMITIOM_BARCODE )
      R_Coil( "GlobalData".FROM_HMI.CTW.RUN_CMD_FROM_HMI )
   END_RUNG
   // the same network as SCL:
   IF "ALARMS".ALARMS.ERROR_8_ERROR_TRANSMITIOM_BARCODE THEN
       "GlobalData".FROM_HMI.CTW.RUN_CMD_FROM_HMI := FALSE;
   END_IF;
END_REGION

REGION Network 8: Сброс ошибки неисправности фотодатчика
   // При появлении сигнала с фотодатчика - сброс ошибки
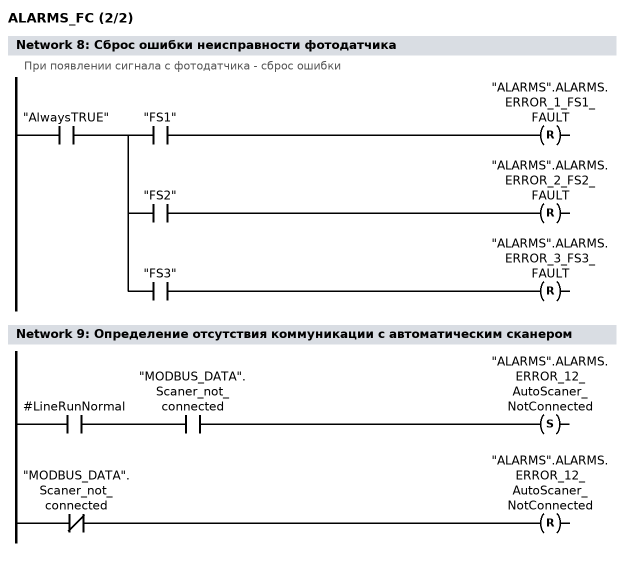
   RUNG wire#powerrail
      Contact( "AlwaysTRUE" )
      wire#w1
      Contact( "FS1" )
      R_Coil( "ALARMS".ALARMS.ERROR_1_FS1_FAULT )
   END_RUNG
   RUNG wire#w1
      Contact( "FS2" )
      R_Coil( "ALARMS".ALARMS.ERROR_2_FS2_FAULT )
   END_RUNG
   RUNG wire#w1
      Contact( "FS3" )
      R_Coil( "ALARMS".ALARMS.ERROR_3_FS3_FAULT )
   END_RUNG
   // the same network as SCL:
   IF "AlwaysTRUE" AND "FS1" THEN "ALARMS".ALARMS.ERROR_1_FS1_FAULT := FALSE; END_IF;
   IF "AlwaysTRUE" AND "FS2" THEN "ALARMS".ALARMS.ERROR_2_FS2_FAULT := FALSE; END_IF;
   IF "AlwaysTRUE" AND "FS3" THEN "ALARMS".ALARMS.ERROR_3_FS3_FAULT := FALSE; END_IF;
END_REGION

REGION Network 9: Определение отсутствия коммуникации с автоматическим сканером
   RUNG wire#powerrail
      Contact( #LineRunNormal )
      Contact( "MODBUS_DATA".Scaner_not_connected )
      S_Coil( "ALARMS".ALARMS.ERROR_12_AutoScaner_NotConnected )
   END_RUNG
   RUNG wire#powerrail
      I_Contact( "MODBUS_DATA".Scaner_not_connected )
      R_Coil( "ALARMS".ALARMS.ERROR_12_AutoScaner_NotConnected )
   END_RUNG
   // the same network as SCL:
   IF #LineRunNormal AND "MODBUS_DATA".Scaner_not_connected THEN
       "ALARMS".ALARMS.ERROR_12_AutoScaner_NotConnected := TRUE;
   END_IF;
   IF NOT "MODBUS_DATA".Scaner_not_connected THEN
       "ALARMS".ALARMS.ERROR_12_AutoScaner_NotConnected := FALSE;
   END_IF;
END_REGION

REGION Network 10 (SCL): Трансфер из битового представления в слово для тэгов HMI
   %DB6.DBW0 := %DB6.DBW4;
   %DB6.DBW2 := %DB6.DBW6;

   %DB6.DBW8 := %DB6.DBW12;
   %DB6.DBW10 := %DB6.DBW14;
END_REGION
END_FUNCTION

// folder: 8_BUZZER

FUNCTION_BLOCK "xBuzzer"   // FB5, LAD
{ S7_Optimized_Access := 'TRUE' }
VERSION : 0.1
   VAR_OUTPUT
      BUZZER_OUT : Bool;
   END_VAR
   VAR_IN_OUT
      IN : Bool;
   END_VAR
   VAR
      "Timer" : TOF_TIME;
      MR0 : Bool;
      RLO_0 : Bool;
   END_VAR
   VAR_TEMP   // added for the SCL form of the ladder/FBD networks
      _w1 : Bool;
   END_VAR
BEGIN

REGION Network 1: Выделение положительного фронта сигнала
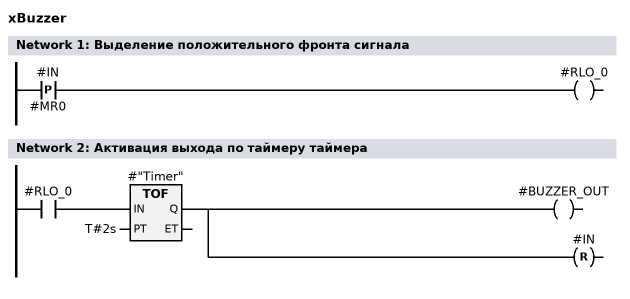
   RUNG wire#powerrail
      P_Contact(operand := #IN, bit := #MR0)
      Coil( #RLO_0 )
   END_RUNG
   // the same network as SCL:
   #_w1 := #IN AND NOT #MR0;   // rising edge of #IN
   #MR0 := #IN;
   #RLO_0 := #_w1;
END_REGION

REGION Network 2: Активация выхода по таймеру таймера
   #"Timer"(IN := #RLO_0, PT := T#2s);   // TOF
   #BUZZER_OUT := #"Timer".Q;
   IF #"Timer".Q THEN #IN := FALSE; END_IF;
END_REGION
END_FUNCTION_BLOCK

// folder: 9_PINOUT

FUNCTION "IO_DEFENITION" : Void   // FC13, LAD
{ S7_Optimized_Access := 'TRUE' }
VERSION : 0.1
   VAR_TEMP
      bEnable : Bool;   // Разрешение
      fs1_state : Bool;   // Инверсный статус FS1
      fs2_state : Bool;   // Инверсный статус FS2
      fs3_state : Bool;   // Инверсный статус FS3
      currentTime : DTL;   // Текущее время
      tmpResult : Int;
   END_VAR
   VAR_TEMP   // added for the SCL form of the ladder/FBD networks
      _w1 : Bool;
   END_VAR
BEGIN

REGION Network 1: Инверсный статус FS1
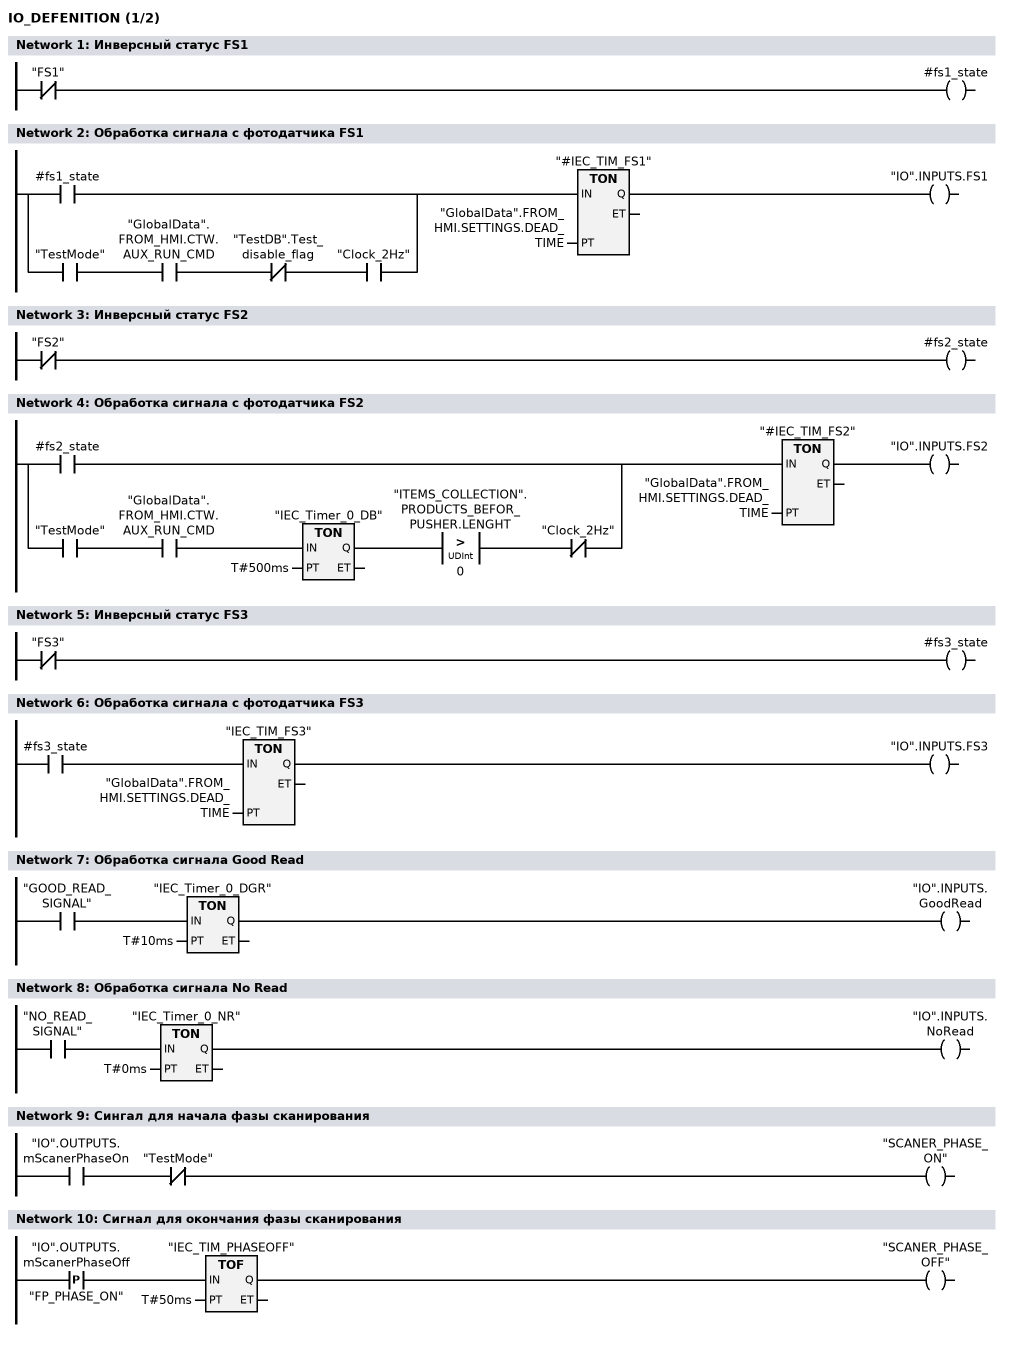
   RUNG wire#powerrail
      I_Contact( "FS1" )
      Coil( #fs1_state )
   END_RUNG
   // the same network as SCL:
   #fs1_state := NOT "FS1";
END_REGION

REGION Network 2: Обработка сигнала с фотодатчика FS1
   "#IEC_TIM_FS1".TON(IN := #fs1_state OR ("TestMode" AND "GlobalData".FROM_HMI.CTW.AUX_RUN_CMD AND NOT "TestDB".Test_disable_flag AND "Clock_2Hz"),
                      PT := "GlobalData".FROM_HMI.SETTINGS.DEAD_TIME);
   "IO".INPUTS.FS1 := "#IEC_TIM_FS1".Q;
END_REGION

REGION Network 3: Инверсный статус FS2
   RUNG wire#powerrail
      I_Contact( "FS2" )
      Coil( #fs2_state )
   END_RUNG
   // the same network as SCL:
   #fs2_state := NOT "FS2";
END_REGION

REGION Network 4: Обработка сигнала с фотодатчика FS2
   "IEC_Timer_0_DB".TON(IN := "TestMode" AND "GlobalData".FROM_HMI.CTW.AUX_RUN_CMD, PT := T#500ms);
   "#IEC_TIM_FS2".TON(IN := #fs2_state OR ("IEC_Timer_0_DB".Q AND ("ITEMS_COLLECTION".PRODUCTS_BEFOR_PUSHER.LENGHT > 0) AND NOT "Clock_2Hz"),
                      PT := "GlobalData".FROM_HMI.SETTINGS.DEAD_TIME);
   "IO".INPUTS.FS2 := "#IEC_TIM_FS2".Q;
END_REGION

REGION Network 5: Инверсный статус FS3
   RUNG wire#powerrail
      I_Contact( "FS3" )
      Coil( #fs3_state )
   END_RUNG
   // the same network as SCL:
   #fs3_state := NOT "FS3";
END_REGION

REGION Network 6: Обработка сигнала с фотодатчика FS3
   "IEC_TIM_FS3".TON(IN := #fs3_state, PT := "GlobalData".FROM_HMI.SETTINGS.DEAD_TIME);
   "IO".INPUTS.FS3 := "IEC_TIM_FS3".Q;
END_REGION

REGION Network 7: Обработка сигнала Good Read
   "IEC_Timer_0_DGR".TON(IN := "GOOD_READ_SIGNAL", PT := T#10ms);
   "IO".INPUTS.GoodRead := "IEC_Timer_0_DGR".Q;
END_REGION

REGION Network 8: Обработка сигнала No Read
   "IEC_Timer_0_NR".TON(IN := "NO_READ_SIGNAL", PT := T#0ms);
   "IO".INPUTS.NoRead := "IEC_Timer_0_NR".Q;
END_REGION

REGION Network 9: Сингал для начала фазы сканирования
   RUNG wire#powerrail
      Contact( "IO".OUTPUTS.mScanerPhaseOn )
      I_Contact( "TestMode" )
      Coil( "SCANER_PHASE_ON" )
   END_RUNG
   // the same network as SCL:
   "SCANER_PHASE_ON" := "IO".OUTPUTS.mScanerPhaseOn AND NOT "TestMode";
END_REGION

REGION Network 10: Сигнал для окончания фазы сканирования
   #_w1 := "IO".OUTPUTS.mScanerPhaseOff AND NOT "FP_PHASE_ON";   // rising edge of "IO".OUTPUTS.mScanerPhaseOff
   "FP_PHASE_ON" := "IO".OUTPUTS.mScanerPhaseOff;
   "IEC_TIM_PHASEOFF".TOF(IN := #_w1, PT := T#50ms);
   "SCANER_PHASE_OFF" := "IEC_TIM_PHASEOFF".Q;
END_REGION

REGION Network 11
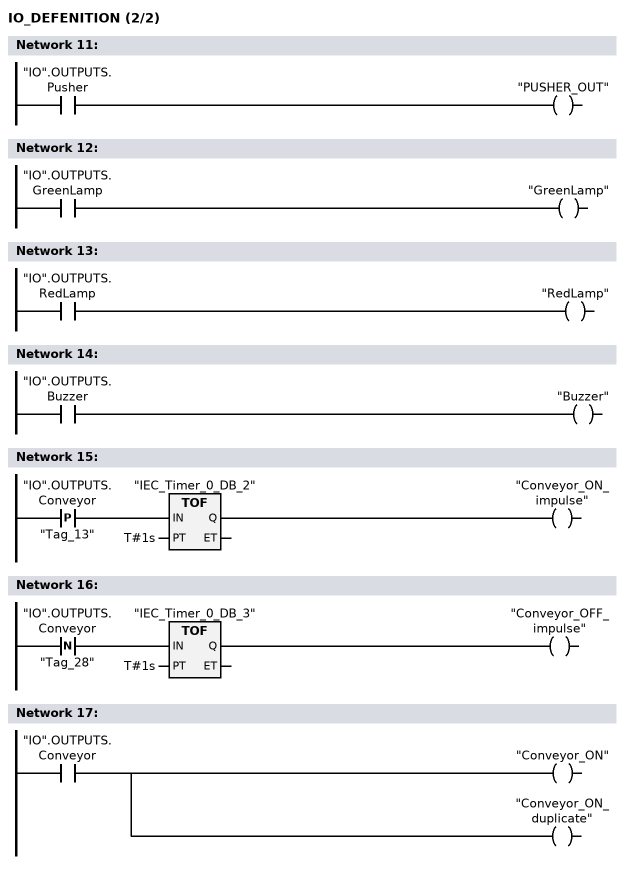
   RUNG wire#powerrail
      Contact( "IO".OUTPUTS.Pusher )
      Coil( "PUSHER_OUT" )
   END_RUNG
   // the same network as SCL:
   "PUSHER_OUT" := "IO".OUTPUTS.Pusher;
END_REGION

REGION Network 12
   RUNG wire#powerrail
      Contact( "IO".OUTPUTS.GreenLamp )
      Coil( "GreenLamp" )
   END_RUNG
   // the same network as SCL:
   "GreenLamp" := "IO".OUTPUTS.GreenLamp;
END_REGION

REGION Network 13
   RUNG wire#powerrail
      Contact( "IO".OUTPUTS.RedLamp )
      Coil( "RedLamp" )
   END_RUNG
   // the same network as SCL:
   "RedLamp" := "IO".OUTPUTS.RedLamp;
END_REGION

REGION Network 14
   RUNG wire#powerrail
      Contact( "IO".OUTPUTS.Buzzer )
      Coil( "Buzzer" )
   END_RUNG
   // the same network as SCL:
   "Buzzer" := "IO".OUTPUTS.Buzzer;
END_REGION

REGION Network 15
   #_w1 := "IO".OUTPUTS.Conveyor AND NOT "Tag_13";   // rising edge of "IO".OUTPUTS.Conveyor
   "Tag_13" := "IO".OUTPUTS.Conveyor;
   "IEC_Timer_0_DB_2".TOF(IN := #_w1, PT := T#1s);
   "Conveyor_ON_impulse" := "IEC_Timer_0_DB_2".Q;
END_REGION

REGION Network 16
   #_w1 := NOT "IO".OUTPUTS.Conveyor AND "Tag_28";   // falling edge of "IO".OUTPUTS.Conveyor
   "Tag_28" := "IO".OUTPUTS.Conveyor;
   "IEC_Timer_0_DB_3".TOF(IN := #_w1, PT := T#1s);
   "Conveyor_OFF_impulse" := "IEC_Timer_0_DB_3".Q;
END_REGION

REGION Network 17
   RUNG wire#powerrail
      Contact( "IO".OUTPUTS.Conveyor )
      wire#w1
      Coil( "Conveyor_ON" )
   END_RUNG
   RUNG wire#w1
      Coil( "Conveyor_ON_duplicate" )
   END_RUNG
   // the same network as SCL:
   "Conveyor_ON" := "IO".OUTPUTS.Conveyor;
   "Conveyor_ON_duplicate" := "IO".OUTPUTS.Conveyor;
END_REGION
END_FUNCTION